LIN {X 0,Y 249.476,Z 748.518,A -85,B 0,C 180,E1 -18809.999,E2 -18809.999} C_VEL
LIN {X 0,Y 249.132,Z 748.626,A -85,B 0,C 180,E1 -18811.616,E2 -18811.616} C_VEL
LIN {X 0,Y 248.499,Z 747.93,A -85,B 0,C 180,E1 -18814.866,E2 -18814.866} C_VEL
LIN {X 0,Y 247.94,Z 746.023,A -85,B 0,C 180,E1 -18818.147,E2 -18818.147} C_VEL
LIN {X 0,Y 247.778,Z 742.93,A -85,B 0,C 180,E1 -18821.451,E2 -18821.451} C_VEL
LIN {X 0,Y 248.292,Z 738.587,A -85,B 0,C 180,E1 -18824.758,E2 -18824.758} C_VEL
LIN {X 0,Y 249.565,Z 732.939,A -85,B 0,C 180,E1 -18828.044,E2 -18828.044} C_VEL
LIN {X 0,Y 251.711,Z 725.892,A -85,B 0,C 180,E1 -18831.282,E2 -18831.282} C_VEL
LIN {X 0,Y 254.679,Z 717.261,A -85,B 0,C 180,E1 -18834.451,E2 -18834.451} C_VEL
LIN {X 0,Y 257.938,Z 708.169,A -85,B 0,C 180,E1 -18837.153,E2 -18837.153} C_VEL
LIN {X 0,Y 261.307,Z 699.031,A -85,B 0,C 180,E1 -18839.395,E2 -18839.395} C_VEL
LIN {X 0,Y 265.243,Z 688.365,A -85,B 0,C 180,E1 -18841.553,E2 -18841.553} C_VEL
LIN {X 0,Y 269.237,Z 676.854,A -85,B 0,C 180,E1 -18843.464,E2 -18843.464} C_VEL
LIN {X 0,Y 273.201,Z 664.412,A -85,B 0,C 180,E1 -18845.139,E2 -18845.139} C_VEL
LIN {X 0,Y 277.197,Z 650.888,A -85,B 0,C 180,E1 -18846.569,E2 -18846.569} C_VEL
LIN {X 0,Y 280.927,Z 635.963,A -85,B 0,C 180,E1 -18847.799,E2 -18847.799} C_VEL
LIN {X 0,Y 283.801,Z 621.53,A -85,B 0,C 180,E1 -18848.701,E2 -18848.701} C_VEL
LIN {X 0,Y 286.017,Z 605.972,A -85,B 0,C 180,E1 -18849.42,E2 -18849.42} C_VEL
LIN {X 0,Y 287.366,Z 589.732,A -85,B 0,C 180,E1 -18849.923,E2 -18849.923} C_VEL
LIN {X 0,Y 290.895,Z 520.508,A -85,B 0,C 180,E1 -18851.589,E2 -18851.589} C_VEL
LIN {X 0,Y 289.329,Z 502.503,A -85,B 0,C 180,E1 -18852.514,E2 -18852.514} C_VEL
LIN {X 0,Y 286.599,Z 477.609,A -85,B 0,C 180,E1 -18853.955,E2 -18853.955} C_VEL
LIN {X 0,Y 285.966,Z 473.872,A -85,B 0,C 180,E1 -18854.225,E2 -18854.225} C_VEL
LIN {X 0,Y 279.058,Z 458.877,A -85,B 0,C 180,E1 -18856.347,E2 -18856.347} C_VEL
LIN {X 0,Y 272.923,Z 447.108,A -85,B 0,C 180,E1 -18858.346,E2 -18858.346} C_VEL
LIN {X 0,Y 268.743,Z 439.718,A -85,B 0,C 180,E1 -18859.789,E2 -18859.789} C_VEL
LIN {X 0,Y 265.068,Z 433.428,A -85,B 0,C 180,E1 -18861.13,E2 -18861.13} C_VEL
LIN {X 0,Y 260.653,Z 426.199,A -85,B 0,C 180,E1 -18862.84,E2 -18862.84} C_VEL
LIN {X 0,Y 256.84,Z 420.001,A -85,B 0,C 180,E1 -18864.446,E2 -18864.446} C_VEL
LIN {X 0,Y 254.494,Z 413.539,A -85,B 0,C 180,E1 -18867.419,E2 -18867.419} C_VEL
LIN {X 0,Y 251.831,Z 406.905,A -85,B 0,C 180,E1 -18870.869,E2 -18870.869} C_VEL
LIN {X 0,Y 249.026,Z 400.088,A -85,B 0,C 180,E1 -18874.956,E2 -18874.956} C_VEL
LIN {X 0,Y 249.041,Z 400.084,A -85,B 0,C 180,E1 -18878.628,E2 -18878.628} C_VEL
LIN {X 0,Y 249.149,Z 400.073,A -85,B 0,C 180,E1 -18883.616,E2 -18883.616} C_VEL
LIN {X 0,Y 249.207,Z 400.066,A -85,B 0,C 180,E1 -18888.615,E2 -18888.615} C_VEL
LIN {X 0,Y 249.42,Z 400.043,A -85,B 0,C 180,E1 -18891.901,E2 -18891.901} C_VEL
LIN {X 0,Y 249.254,Z 400.062,A -85,B 0,C 180,E1 -18895.148,E2 -18895.148} C_VEL
LIN {X 0,Y 249.647,Z 400.005,A -85,B 0,C 180,E1 -18898.387,E2 -18898.387} C_VEL
LIN {X 0,Y 249.651,Z 400.002,A -85,B 0,C 180,E1 -18901.614,E2 -18901.614} C_VEL
LIN {X 0,Y 249.397,Z 399.996,A -85,B 0,C 180,E1 -18906.735,E2 -18906.735} C_VEL
LIN {X 0,Y 249.324,Z 400.04,A -85,B 0,C 180,E1 -18909.738,E2 -18909.738} C_VEL
LIN {X 0,Y 249.169,Z 400.033,A -85,B 0,C 180,E1 -18914.706,E2 -18914.706} C_VEL
LIN {X 0,Y 249.103,Z 400.079,A -85,B 0,C 180,E1 -18918.08,E2 -18918.08} C_VEL
LIN {X 0,Y 249.07,Z 400.051,A -85,B 0,C 180,E1 -18921.52,E2 -18921.52} C_VEL
LIN {X 0,Y 249.057,Z 400.222,A -85,B 0,C 180,E1 -18924.486,E2 -18924.486} C_VEL
LIN {X 0,Y 249.847,Z 402.583,A -85,B 0,C 180,E1 -18924.958,E2 -18924.958} C_VEL
LIN {X 0,Y 251.68,Z 404.775,A -85,B 0,C 180,E1 -18925.83,E2 -18925.83} C_VEL
LIN {X 0,Y 253.402,Z 405.892,A -85,B 0,C 180,E1 -18926.566,E2 -18926.566} C_VEL
LIN {X 0,Y 255.21,Z 409.013,A -85,B 0,C 180,E1 -18927.414,E2 -18927.414} C_VEL
LIN {X 0,Y 257.729,Z 411.478,A -85,B 0,C 180,E1 -18928.445,E2 -18928.445} C_VEL
LIN {X 0,Y 260.121,Z 414.887,A -85,B 0,C 180,E1 -18929.433,E2 -18929.433} C_VEL
LIN {X 0,Y 261.868,Z 416.787,A -85,B 0,C 180,E1 -18930.099,E2 -18930.099} C_VEL
LIN {X 0,Y 264.729,Z 420.479,A -85,B 0,C 180,E1 -18931.174,E2 -18931.174} C_VEL
LIN {X 0,Y 269.59,Z 427.111,A -85,B 0,C 180,E1 -18932.901,E2 -18932.901} C_VEL
LIN {X 0,Y 274.586,Z 434.03,A -85,B 0,C 180,E1 -18934.548,E2 -18934.548} C_VEL
LIN {X 0,Y 283.18,Z 447.173,A -85,B 0,C 180,E1 -18937.169,E2 -18937.169} C_VEL
LIN {X 0,Y 291.353,Z 460.987,A -85,B 0,C 180,E1 -18939.448,E2 -18939.448} C_VEL
LIN {X 0,Y 293.531,Z 464.988,A -85,B 0,C 180,E1 -18940.029,E2 -18940.029} C_VEL
LIN {X 0,Y 290.894,Z 517.972,A -85,B 0,C 180,E1 -18941.323,E2 -18941.323} C_VEL
LIN {X 0,Y 289.972,Z 539.395,A -85,B 0,C 180,E1 -18941.982,E2 -18941.982} C_VEL
LIN {X 0,Y 288.744,Z 554.324,A -85,B 0,C 180,E1 -18942.716,E2 -18942.716} C_VEL
LIN {X 0,Y 286.941,Z 567.715,A -85,B 0,C 180,E1 -18943.579,E2 -18943.579} C_VEL
LIN {X 0,Y 284.605,Z 581.657,A -85,B 0,C 180,E1 -18944.772,E2 -18944.772} C_VEL
LIN {X 0,Y 281.516,Z 595.873,A -85,B 0,C 180,E1 -18946.303,E2 -18946.303} C_VEL
LIN {X 0,Y 278.175,Z 608.428,A -85,B 0,C 180,E1 -18947.973,E2 -18947.973} C_VEL
LIN {X 0,Y 274.87,Z 619.546,A -85,B 0,C 180,E1 -18949.791,E2 -18949.791} C_VEL
LIN {X 0,Y 271.101,Z 630.65,A -85,B 0,C 180,E1 -18952,E2 -18952} C_VEL
LIN {X 0,Y 267.58,Z 639.923,A -85,B 0,C 180,E1 -18954.241,E2 -18954.241} C_VEL
LIN {X 0,Y 263.922,Z 648.935,A -85,B 0,C 180,E1 -18956.916,E2 -18956.916} C_VEL
LIN {X 0,Y 260.559,Z 656.451,A -85,B 0,C 180,E1 -18959.671,E2 -18959.671} C_VEL
LIN {X 0,Y 257.771,Z 662.395,A -85,B 0,C 180,E1 -18962.388,E2 -18962.388} C_VEL
LIN {X 0,Y 255.141,Z 667.863,A -85,B 0,C 180,E1 -18965.596,E2 -18965.596} C_VEL
LIN {X 0,Y 252.997,Z 671.949,A -85,B 0,C 180,E1 -18968.832,E2 -18968.832} C_VEL
LIN {X 0,Y 251.419,Z 674.771,A -85,B 0,C 180,E1 -18972.093,E2 -18972.093} C_VEL
LIN {X 0,Y 250.317,Z 676.423,A -85,B 0,C 180,E1 -18975.364,E2 -18975.364} C_VEL
LIN {X 0,Y 249.779,Z 676.905,A -85,B 0,C 180,E1 -18978.642,E2 -18978.642} C_VEL
LIN {X 0,Y 249.622,Z 676.258,A -85,B 0,C 180,E1 -18981.908,E2 -18981.908} C_VEL
LIN {X 0,Y 249.657,Z 674.55,A -85,B 0,C 180,E1 -18985.156,E2 -18985.156} C_VEL
LIN {X 0,Y 250.221,Z 671.7,A -85,B 0,C 180,E1 -18988.391,E2 -18988.391} C_VEL
LIN {X 0,Y 251.252,Z 667.656,A -85,B 0,C 180,E1 -18991.603,E2 -18991.603} C_VEL
LIN {X 0,Y 252.64,Z 662.347,A -85,B 0,C 180,E1 -18994.788,E2 -18994.788} C_VEL
LIN {X 0,Y 254.541,Z 655.601,A -85,B 0,C 180,E1 -18997.936,E2 -18997.936} C_VEL
LIN {X 0,Y 256.823,Z 647.225,A -85,B 0,C 180,E1 -19001.044,E2 -19001.044} C_VEL
LIN {X 0,Y 259.301,Z 638.318,A -85,B 0,C 180,E1 -19003.719,E2 -19003.719} C_VEL
LIN {X 0,Y 261.672,Z 629.26,A -85,B 0,C 180,E1 -19005.98,E2 -19005.98} C_VEL
LIN {X 0,Y 264.275,Z 618.53,A -85,B 0,C 180,E1 -19008.208,E2 -19008.208} C_VEL
LIN {X 0,Y 266.7,Z 606.853,A -85,B 0,C 180,E1 -19010.235,E2 -19010.235} C_VEL
LIN {X 0,Y 269.276,Z 594.003,A -85,B 0,C 180,E1 -19012.036,E2 -19012.036} C_VEL
LIN {X 0,Y 271.443,Z 581.475,A -85,B 0,C 180,E1 -19013.458,E2 -19013.458} C_VEL
LIN {X 0,Y 273.344,Z 567.926,A -85,B 0,C 180,E1 -19014.696,E2 -19014.696} C_VEL
LIN {X 0,Y 274.933,Z 552.816,A -85,B 0,C 180,E1 -19015.757,E2 -19015.757} C_VEL
LIN {X 0,Y 276.006,Z 537.572,A -85,B 0,C 180,E1 -19016.522,E2 -19016.522} C_VEL
LIN {X 0,Y 276.531,Z 519.72,A -85,B 0,C 180,E1 -19017.106,E2 -19017.106} C_VEL
LIN {X 0,Y 279.032,Z 452.977,A -85,B 0,C 180,E1 -19018.811,E2 -19018.811} C_VEL
LIN {X 0,Y 270.28,Z 435.589,A -85,B 0,C 180,E1 -19020.695,E2 -19020.695} C_VEL
LIN {X 0,Y 260.936,Z 419.389,A -85,B 0,C 180,E1 -19022.818,E2 -19022.818} C_VEL
LIN {X 0,Y 253.534,Z 407.906,A -85,B 0,C 180,E1 -19024.61,E2 -19024.61} C_VEL
LIN {X 0,Y 251.344,Z 404.489,A -85,B 0,C 180,E1 -19025.171,E2 -19025.171} C_VEL
LIN {X 0,Y 249.599,Z 402.156,A -85,B 0,C 180,E1 -19025.614,E2 -19025.614} C_VEL
LIN {X 0,Y 249.025,Z 400.089,A -85,B 0,C 180,E1 -19025.851,E2 -19025.851} C_VEL
LIN {X 0,Y 249.012,Z 400.093,A -85,B 0,C 180,E1 -19028.383,E2 -19028.383} C_VEL
LIN {X 0,Y 248.956,Z 400.094,A -85,B 0,C 180,E1 -19032.778,E2 -19032.778} C_VEL
LIN {X 0,Y 248.966,Z 400.089,A -85,B 0,C 180,E1 -19037.352,E2 -19037.352} C_VEL
LIN {X 0,Y 249.001,Z 400.085,A -85,B 0,C 180,E1 -19041.614,E2 -19041.614} C_VEL
LIN {X 0,Y 249.041,Z 400.079,A -85,B 0,C 180,E1 -19045.638,E2 -19045.638} C_VEL
LIN {X 0,Y 248.991,Z 400.093,A -85,B 0,C 180,E1 -19049.464,E2 -19049.464} C_VEL
LIN {X 0,Y 249.02,Z 400.093,A -85,B 0,C 180,E1 -19053.156,E2 -19053.156} C_VEL
LIN {X 0,Y 249.048,Z 400.077,A -85,B 0,C 180,E1 -19056.729,E2 -19056.729} C_VEL
LIN {X 0,Y 249.044,Z 400.08,A -85,B 0,C 180,E1 -19060.206,E2 -19060.206} C_VEL
LIN {X 0,Y 249.155,Z 400.076,A -85,B 0,C 180,E1 -19063.616,E2 -19063.616} C_VEL
LIN {X 0,Y 249.181,Z 400.035,A -85,B 0,C 180,E1 -19066.959,E2 -19066.959} C_VEL
LIN {X 0,Y 249.367,Z 399.996,A -85,B 0,C 180,E1 -19070.599,E2 -19070.599} C_VEL
LIN {X 0,Y 249.414,Z 400.036,A -85,B 0,C 180,E1 -19073.528,E2 -19073.528} C_VEL
LIN {X 0,Y 249.476,Z 400.016,A -85,B 0,C 180,E1 -19077.599,E2 -19077.599} C_VEL
LIN {X 0,Y 248.956,Z 400.086,A -85,B 0,C 180,E1 -19078.948,E2 -19078.948} C_VEL
LIN {X 0,Y 247.373,Z 400.295,A -85,B 0,C 180,E1 -19080.27,E2 -19080.27} C_VEL
LIN {X 0,Y 243.446,Z 400.774,A -85,B 0,C 180,E1 -19082.93,E2 -19082.93} C_VEL
LIN {X 0,Y 242.313,Z 400.91,A -85,B 0,C 180,E1 -19084.323,E2 -19084.323} C_VEL
LIN {X 0,Y 242.218,Z 400.925,A -85,B 0,C 180,E1 -19084.796,E2 -19084.796} C_VEL
LIN {X 0,Y 242.389,Z 400.915,A -85,B 0,C 180,E1 -19086.66,E2 -19086.66} C_VEL
LIN {X 0,Y 242.256,Z 400.921,A -85,B 0,C 180,E1 -19090.024,E2 -19090.024} C_VEL
LIN {X 0,Y 242.098,Z 400.944,A -85,B 0,C 180,E1 -19095.145,E2 -19095.145} C_VEL
LIN {X 0,Y 242.009,Z 400.954,A -85,B 0,C 180,E1 -19098.629,E2 -19098.629} C_VEL
LIN {X 0,Y 241.969,Z 400.963,A -85,B 0,C 180,E1 -19102.184,E2 -19102.184} C_VEL
LIN {X 0,Y 241.983,Z 400.962,A -85,B 0,C 180,E1 -19105.826,E2 -19105.826} C_VEL
LIN {X 0,Y 241.959,Z 400.966,A -85,B 0,C 180,E1 -19109.589,E2 -19109.589} C_VEL
LIN {X 0,Y 241.975,Z 400.948,A -85,B 0,C 180,E1 -19113.493,E2 -19113.493} C_VEL
LIN {X 0,Y 241.995,Z 401.064,A -85,B 0,C 180,E1 -19115.509,E2 -19115.509} C_VEL
LIN {X 0,Y 246.124,Z 413.213,A -85,B 0,C 180,E1 -19119.976,E2 -19119.976} C_VEL
LIN {X 0,Y 249.086,Z 422.878,A -85,B 0,C 180,E1 -19123.174,E2 -19123.174} C_VEL
LIN {X 0,Y 250.292,Z 426.911,A -85,B 0,C 180,E1 -19124.374,E2 -19124.374} C_VEL
LIN {X 0,Y 258.143,Z 443.198,A -85,B 0,C 180,E1 -19126.434,E2 -19126.434} C_VEL
LIN {X 0,Y 264.737,Z 458.633,A -85,B 0,C 180,E1 -19128.09,E2 -19128.09} C_VEL
LIN {X 0,Y 265.62,Z 461.45,A -85,B 0,C 180,E1 -19128.327,E2 -19128.327} C_VEL
LIN {X 0,Y 268.764,Z 492.72,A -85,B 0,C 180,E1 -19129.844,E2 -19129.844} C_VEL
LIN {X 0,Y 271.266,Z 519.191,A -85,B 0,C 180,E1 -19131.056,E2 -19131.056} C_VEL
LIN {X 0,Y 267.769,Z 598.776,A -85,B 0,C 180,E1 -19133.103,E2 -19133.103} C_VEL
LIN {X 0,Y 266.362,Z 614.419,A -85,B 0,C 180,E1 -19133.759,E2 -19133.759} C_VEL
LIN {X 0,Y 264.285,Z 629.484,A -85,B 0,C 180,E1 -19134.663,E2 -19134.663} C_VEL
LIN {X 0,Y 261.597,Z 644.604,A -85,B 0,C 180,E1 -19135.888,E2 -19135.888} C_VEL
LIN {X 0,Y 258.665,Z 657.774,A -85,B 0,C 180,E1 -19137.253,E2 -19137.253} C_VEL
LIN {X 0,Y 256.507,Z 666.573,A -85,B 0,C 180,E1 -19138.353,E2 -19138.353} C_VEL
LIN {X 0,Y 253.528,Z 679.329,A -85,B 0,C 180,E1 -19140.297,E2 -19140.297} C_VEL
LIN {X 0,Y 250.464,Z 690.836,A -85,B 0,C 180,E1 -19142.42,E2 -19142.42} C_VEL
LIN {X 0,Y 247.407,Z 702.532,A -85,B 0,C 180,E1 -19145.081,E2 -19145.081} C_VEL
LIN {X 0,Y 245.08,Z 711.881,A -85,B 0,C 180,E1 -19147.669,E2 -19147.669} C_VEL
LIN {X 0,Y 243.175,Z 720.586,A -85,B 0,C 180,E1 -19150.588,E2 -19150.588} C_VEL
LIN {X 0,Y 241.833,Z 727.828,A -85,B 0,C 180,E1 -19153.54,E2 -19153.54} C_VEL
LIN {X 0,Y 241.125,Z 733.822,A -85,B 0,C 180,E1 -19156.516,E2 -19156.516} C_VEL
LIN {X 0,Y 240.966,Z 739.281,A -85,B 0,C 180,E1 -19159.921,E2 -19159.921} C_VEL
LIN {X 0,Y 241.306,Z 743.356,A -85,B 0,C 180,E1 -19163.309,E2 -19163.309} C_VEL
LIN {X 0,Y 241.603,Z 744.896,A -85,B 0,C 180,E1 -19164.993,E2 -19164.993} C_VEL
LIN {X 0,Y 242.142,Z 746.94,A -85,B 0,C 180,E1 -19168.336,E2 -19168.336} C_VEL
LIN {X 0,Y 242.448,Z 747.474,A -85,B 0,C 180,E1 -19169.999,E2 -19169.999} C_VEL
LIN {X 0,Y 242.093,Z 747.598,A -85,B 0,C 180,E1 -19171.663,E2 -19171.663} C_VEL
LIN {X 0,Y 241.409,Z 746.93,A -85,B 0,C 180,E1 -19175.01,E2 -19175.01} C_VEL
LIN {X 0,Y 240.834,Z 745.054,A -85,B 0,C 180,E1 -19178.389,E2 -19178.389} C_VEL
LIN {X 0,Y 240.725,Z 741.993,A -85,B 0,C 180,E1 -19181.791,E2 -19181.791} C_VEL
LIN {X 0,Y 241.338,Z 737.677,A -85,B 0,C 180,E1 -19185.193,E2 -19185.193} C_VEL
LIN {X 0,Y 242.69,Z 732.068,A -85,B 0,C 180,E1 -19188.574,E2 -19188.574} C_VEL
LIN {X 0,Y 244.997,Z 725.073,A -85,B 0,C 180,E1 -19191.894,E2 -19191.894} C_VEL
LIN {X 0,Y 248.143,Z 716.501,A -85,B 0,C 180,E1 -19195.139,E2 -19195.139} C_VEL
LIN {X 0,Y 251.56,Z 707.476,A -85,B 0,C 180,E1 -19197.9,E2 -19197.9} C_VEL
LIN {X 0,Y 255.108,Z 698.413,A -85,B 0,C 180,E1 -19200.182,E2 -19200.182} C_VEL
LIN {X 0,Y 259.19,Z 687.83,A -85,B 0,C 180,E1 -19202.378,E2 -19202.378} C_VEL
LIN {X 0,Y 263.683,Z 675.235,A -85,B 0,C 180,E1 -19204.496,E2 -19204.496} C_VEL
LIN {X 0,Y 267.847,Z 662.7,A -85,B 0,C 180,E1 -19206.182,E2 -19206.182} C_VEL
LIN {X 0,Y 271.983,Z 649.046,A -85,B 0,C 180,E1 -19207.621,E2 -19207.621} C_VEL
LIN {X 0,Y 275.601,Z 634.964,A -85,B 0,C 180,E1 -19208.78,E2 -19208.78} C_VEL
LIN {X 0,Y 278.558,Z 620.543,A -85,B 0,C 180,E1 -19209.688,E2 -19209.688} C_VEL
LIN {X 0,Y 280.72,Z 605.925,A -85,B 0,C 180,E1 -19210.374,E2 -19210.374} C_VEL
LIN {X 0,Y 282.138,Z 590.291,A -85,B 0,C 180,E1 -19210.879,E2 -19210.879} C_VEL
LIN {X 0,Y 285.805,Z 521.741,A -85,B 0,C 180,E1 -19212.551,E2 -19212.551} C_VEL
LIN {X 0,Y 284.506,Z 505.394,A -85,B 0,C 180,E1 -19213.399,E2 -19213.399} C_VEL
LIN {X 0,Y 281.744,Z 479.095,A -85,B 0,C 180,E1 -19214.959,E2 -19214.959} C_VEL
LIN {X 0,Y 281.208,Z 476.865,A -85,B 0,C 180,E1 -19215.163,E2 -19215.163} C_VEL
LIN {X 0,Y 275.137,Z 463.465,A -85,B 0,C 180,E1 -19217.118,E2 -19217.118} C_VEL
LIN {X 0,Y 268.864,Z 451.319,A -85,B 0,C 180,E1 -19219.255,E2 -19219.255} C_VEL
LIN {X 0,Y 265.135,Z 444.539,A -85,B 0,C 180,E1 -19220.608,E2 -19220.608} C_VEL
LIN {X 0,Y 261.817,Z 438.739,A -85,B 0,C 180,E1 -19221.874,E2 -19221.874} C_VEL
LIN {X 0,Y 257.664,Z 431.782,A -85,B 0,C 180,E1 -19223.552,E2 -19223.552} C_VEL
LIN {X 0,Y 253.275,Z 424.794,A -85,B 0,C 180,E1 -19225.46,E2 -19225.46} C_VEL
LIN {X 0,Y 248.719,Z 417.542,A -85,B 0,C 180,E1 -19227.679,E2 -19227.679} C_VEL
LIN {X 0,Y 246.271,Z 411.332,A -85,B 0,C 180,E1 -19230.979,E2 -19230.979} C_VEL
LIN {X 0,Y 243.388,Z 404.393,A -85,B 0,C 180,E1 -19235.248,E2 -19235.248} C_VEL
LIN {X 0,Y 241.947,Z 401.013,A -85,B 0,C 180,E1 -19237.646,E2 -19237.646} C_VEL
LIN {X 0,Y 242.002,Z 400.965,A -85,B 0,C 180,E1 -19241.371,E2 -19241.371} C_VEL
LIN {X 0,Y 242.093,Z 400.954,A -85,B 0,C 180,E1 -19244.855,E2 -19244.855} C_VEL
LIN {X 0,Y 242.317,Z 400.917,A -85,B 0,C 180,E1 -19250.427,E2 -19250.427} C_VEL
LIN {X 0,Y 242.389,Z 400.906,A -85,B 0,C 180,E1 -19253.34,E2 -19253.34} C_VEL
LIN {X 0,Y 242.607,Z 400.882,A -85,B 0,C 180,E1 -19258.34,E2 -19258.34} C_VEL
LIN {X 0,Y 242.611,Z 400.878,A -85,B 0,C 180,E1 -19261.66,E2 -19261.66} C_VEL
LIN {X 0,Y 242.38,Z 400.87,A -85,B 0,C 180,E1 -19266.705,E2 -19266.705} C_VEL
LIN {X 0,Y 242.253,Z 400.925,A -85,B 0,C 180,E1 -19270.025,E2 -19270.025} C_VEL
LIN {X 0,Y 242.127,Z 400.911,A -85,B 0,C 180,E1 -19275.144,E2 -19275.144} C_VEL
LIN {X 0,Y 242.04,Z 400.947,A -85,B 0,C 180,E1 -19278.627,E2 -19278.627} C_VEL
LIN {X 0,Y 242.033,Z 400.966,A -85,B 0,C 180,E1 -19281.288,E2 -19281.288} C_VEL
LIN {X 0,Y 242.847,Z 403.534,A -85,B 0,C 180,E1 -19281.866,E2 -19281.866} C_VEL
LIN {X 0,Y 244.758,Z 405.758,A -85,B 0,C 180,E1 -19282.92,E2 -19282.92} C_VEL
LIN {X 0,Y 246.638,Z 406.982,A -85,B 0,C 180,E1 -19283.846,E2 -19283.846} C_VEL
LIN {X 0,Y 248.47,Z 410.136,A -85,B 0,C 180,E1 -19284.826,E2 -19284.826} C_VEL
LIN {X 0,Y 251.111,Z 412.591,A -85,B 0,C 180,E1 -19286.045,E2 -19286.045} C_VEL
LIN {X 0,Y 253.503,Z 415.98,A -85,B 0,C 180,E1 -19287.153,E2 -19287.153} C_VEL
LIN {X 0,Y 255.422,Z 418.046,A -85,B 0,C 180,E1 -19287.966,E2 -19287.966} C_VEL
LIN {X 0,Y 257.975,Z 421.43,A -85,B 0,C 180,E1 -19289.034,E2 -19289.034} C_VEL
LIN {X 0,Y 259.356,Z 423.134,A -85,B 0,C 180,E1 -19289.584,E2 -19289.584} C_VEL
LIN {X 0,Y 263.088,Z 428.119,A -85,B 0,C 180,E1 -19291.022,E2 -19291.022} C_VEL
LIN {X 0,Y 266.703,Z 433.046,A -85,B 0,C 180,E1 -19292.334,E2 -19292.334} C_VEL
LIN {X 0,Y 271.875,Z 440.463,A -85,B 0,C 180,E1 -19294.099,E2 -19294.099} C_VEL
LIN {X 0,Y 279.124,Z 451.673,A -85,B 0,C 180,E1 -19296.389,E2 -19296.389} C_VEL
LIN {X 0,Y 287.093,Z 465.293,A -85,B 0,C 180,E1 -19298.706,E2 -19298.706} C_VEL
LIN {X 0,Y 288.491,Z 467.862,A -85,B 0,C 180,E1 -19299.096,E2 -19299.096} C_VEL
LIN {X 0,Y 285.88,Z 517.389,A -85,B 0,C 180,E1 -19300.309,E2 -19300.309} C_VEL
LIN {X 0,Y 284.888,Z 539.899,A -85,B 0,C 180,E1 -19301.001,E2 -19301.001} C_VEL
LIN {X 0,Y 283.666,Z 554.622,A -85,B 0,C 180,E1 -19301.726,E2 -19301.726} C_VEL
LIN {X 0,Y 281.799,Z 568.179,A -85,B 0,C 180,E1 -19302.597,E2 -19302.597} C_VEL
LIN {X 0,Y 279.545,Z 581.338,A -85,B 0,C 180,E1 -19303.716,E2 -19303.716} C_VEL
LIN {X 0,Y 276.494,Z 595.225,A -85,B 0,C 180,E1 -19305.194,E2 -19305.194} C_VEL
LIN {X 0,Y 272.871,Z 608.583,A -85,B 0,C 180,E1 -19306.961,E2 -19306.961} C_VEL
LIN {X 0,Y 269.36,Z 619.805,A -85,B 0,C 180,E1 -19308.793,E2 -19308.793} C_VEL
LIN {X 0,Y 265.429,Z 631.04,A -85,B 0,C 180,E1 -19311.037,E2 -19311.037} C_VEL
LIN {X 0,Y 261.182,Z 641.842,A -85,B 0,C 180,E1 -19313.704,E2 -19313.704} C_VEL
LIN {X 0,Y 257.375,Z 650.701,A -85,B 0,C 180,E1 -19316.432,E2 -19316.432} C_VEL
LIN {X 0,Y 253.832,Z 658.261,A -85,B 0,C 180,E1 -19319.322,E2 -19319.322} C_VEL
LIN {X 0,Y 250.647,Z 664.691,A -85,B 0,C 180,E1 -19322.443,E2 -19322.443} C_VEL
LIN {X 0,Y 247.981,Z 669.856,A -85,B 0,C 180,E1 -19325.737,E2 -19325.737} C_VEL
LIN {X 0,Y 246.308,Z 672.817,A -85,B 0,C 180,E1 -19328.228,E2 -19328.228} C_VEL
LIN {X 0,Y 244.592,Z 675.7,A -85,B 0,C 180,E1 -19331.576,E2 -19331.576} C_VEL
LIN {X 0,Y 243.415,Z 677.401,A -85,B 0,C 180,E1 -19334.94,E2 -19334.94} C_VEL
LIN {X 0,Y 242.789,Z 677.917,A -85,B 0,C 180,E1 -19338.31,E2 -19338.31} C_VEL
LIN {X 0,Y 242.603,Z 677.323,A -85,B 0,C 180,E1 -19341.673,E2 -19341.673} C_VEL
LIN {X 0,Y 242.611,Z 675.672,A -85,B 0,C 180,E1 -19345.015,E2 -19345.015} C_VEL
LIN {X 0,Y 243.18,Z 672.879,A -85,B 0,C 180,E1 -19348.345,E2 -19348.345} C_VEL
LIN {X 0,Y 244.253,Z 668.892,A -85,B 0,C 180,E1 -19351.649,E2 -19351.649} C_VEL
LIN {X 0,Y 245.656,Z 663.651,A -85,B 0,C 180,E1 -19354.924,E2 -19354.924} C_VEL
LIN {X 0,Y 247.619,Z 656.972,A -85,B 0,C 180,E1 -19358.159,E2 -19358.159} C_VEL
LIN {X 0,Y 249.975,Z 648.679,A -85,B 0,C 180,E1 -19361.35,E2 -19361.35} C_VEL
LIN {X 0,Y 252.529,Z 639.858,A -85,B 0,C 180,E1 -19364.094,E2 -19364.094} C_VEL
LIN {X 0,Y 255.422,Z 629.232,A -85,B 0,C 180,E1 -19366.793,E2 -19366.793} C_VEL
LIN {X 0,Y 258.142,Z 618.335,A -85,B 0,C 180,E1 -19369.069,E2 -19369.069} C_VEL
LIN {X 0,Y 260.727,Z 606.417,A -85,B 0,C 180,E1 -19371.133,E2 -19371.133} C_VEL
LIN {X 0,Y 263.482,Z 593.234,A -85,B 0,C 180,E1 -19372.961,E2 -19372.961} C_VEL
LIN {X 0,Y 265.601,Z 580.35,A -85,B 0,C 180,E1 -19374.422,E2 -19374.422} C_VEL
LIN {X 0,Y 267.634,Z 566.182,A -85,B 0,C 180,E1 -19375.676,E2 -19375.676} C_VEL
LIN {X 0,Y 269.175,Z 551.454,A -85,B 0,C 180,E1 -19376.673,E2 -19376.673} C_VEL
LIN {X 0,Y 270.191,Z 536.263,A -85,B 0,C 180,E1 -19377.406,E2 -19377.406} C_VEL
LIN {X 0,Y 270.913,Z 511.116,A -85,B 0,C 180,E1 -19378.168,E2 -19378.168} C_VEL
LIN {X 0,Y 273.171,Z 455.24,A -85,B 0,C 180,E1 -19379.609,E2 -19379.609} C_VEL
LIN {X 0,Y 264.991,Z 438.961,A -85,B 0,C 180,E1 -19381.448,E2 -19381.448} C_VEL
LIN {X 0,Y 256.254,Z 423.785,A -85,B 0,C 180,E1 -19383.515,E2 -19383.515} C_VEL
LIN {X 0,Y 249.341,Z 412.874,A -85,B 0,C 180,E1 -19385.261,E2 -19385.261} C_VEL
LIN {X 0,Y 246.808,Z 409.184,A -85,B 0,C 180,E1 -19385.925,E2 -19385.925} C_VEL
LIN {X 0,Y 244.539,Z 405.59,A -85,B 0,C 180,E1 -19386.549,E2 -19386.549} C_VEL
LIN {X 0,Y 242.615,Z 403.171,A -85,B 0,C 180,E1 -19387.066,E2 -19387.066} C_VEL
LIN {X 0,Y 241.977,Z 400.963,A -85,B 0,C 180,E1 -19387.31,E2 -19387.31} C_VEL
LIN {X 0,Y 241.898,Z 400.979,A -85,B 0,C 180,E1 -19391.93,E2 -19391.93} C_VEL
LIN {X 0,Y 241.892,Z 400.974,A -85,B 0,C 180,E1 -19396.581,E2 -19396.581} C_VEL
LIN {X 0,Y 241.973,Z 400.96,A -85,B 0,C 180,E1 -19401.646,E2 -19401.646} C_VEL
LIN {X 0,Y 241.972,Z 400.971,A -85,B 0,C 180,E1 -19404.486,E2 -19404.486} C_VEL
LIN {X 0,Y 241.946,Z 400.974,A -85,B 0,C 180,E1 -19408.475,E2 -19408.475} C_VEL
LIN {X 0,Y 241.953,Z 400.969,A -85,B 0,C 180,E1 -19412.305,E2 -19412.305} C_VEL
LIN {X 0,Y 242.019,Z 400.95,A -85,B 0,C 180,E1 -19416.011,E2 -19416.011} C_VEL
LIN {X 0,Y 241.984,Z 400.963,A -85,B 0,C 180,E1 -19419.603,E2 -19419.603} C_VEL
LIN {X 0,Y 242.111,Z 400.951,A -85,B 0,C 180,E1 -19423.317,E2 -19423.317} C_VEL
LIN {X 0,Y 242.157,Z 400.888,A -85,B 0,C 180,E1 -19428.278,E2 -19428.278} C_VEL
LIN {X 0,Y 242.353,Z 400.886,A -85,B 0,C 180,E1 -19431.663,E2 -19431.663} C_VEL
LIN {X 0,Y 242.384,Z 400.91,A -85,B 0,C 180,E1 -19433.339,E2 -19433.339} C_VEL
LIN {X 0,Y 242.602,Z 400.872,A -85,B 0,C 180,E1 -19438.34,E2 -19438.34} C_VEL
LIN {X 0,Y 242.612,Z 400.885,A -85,B 0,C 180,E1 -19441.66,E2 -19441.66} C_VEL
LIN {X 0,Y 242.218,Z 400.925,A -85,B 0,C 180,E1 -19444.796,E2 -19444.796} C_VEL
LIN {X 0,Y 241.548,Z 401.021,A -85,B 0,C 180,E1 -19446.186,E2 -19446.186} C_VEL
LIN {X 0,Y 238.708,Z 401.391,A -85,B 0,C 180,E1 -19448.454,E2 -19448.454} C_VEL
LIN {X 0,Y 235.431,Z 401.792,A -85,B 0,C 180,E1 -19451.251,E2 -19451.251} C_VEL
LIN {X 0,Y 235.067,Z 401.827,A -85,B 0,C 180,E1 -19452.22,E2 -19452.22} C_VEL
LIN {X 0,Y 235.046,Z 401.833,A -85,B 0,C 180,E1 -19456.902,E2 -19456.902} C_VEL
LIN {X 0,Y 234.954,Z 401.838,A -85,B 0,C 180,E1 -19461.987,E2 -19461.987} C_VEL
LIN {X 0,Y 234.901,Z 401.843,A -85,B 0,C 180,E1 -19466.665,E2 -19466.665} C_VEL
LIN {X 0,Y 234.891,Z 401.851,A -85,B 0,C 180,E1 -19470.573,E2 -19470.573} C_VEL
LIN {X 0,Y 234.991,Z 402.02,A -85,B 0,C 180,E1 -19474.204,E2 -19474.204} C_VEL
LIN {X 0,Y 238.526,Z 412.295,A -85,B 0,C 180,E1 -19478.224,E2 -19478.224} C_VEL
LIN {X 0,Y 241.857,Z 422.842,A -85,B 0,C 180,E1 -19481.939,E2 -19481.939} C_VEL
LIN {X 0,Y 242.672,Z 425.504,A -85,B 0,C 180,E1 -19482.75,E2 -19482.75} C_VEL
LIN {X 0,Y 249.12,Z 438.303,A -85,B 0,C 180,E1 -19484.568,E2 -19484.568} C_VEL
LIN {X 0,Y 255.679,Z 452.618,A -85,B 0,C 180,E1 -19486.324,E2 -19486.324} C_VEL
LIN {X 0,Y 260.042,Z 463.529,A -85,B 0,C 180,E1 -19487.471,E2 -19487.471} C_VEL
LIN {X 0,Y 263.043,Z 494.261,A -85,B 0,C 180,E1 -19489.004,E2 -19489.004} C_VEL
LIN {X 0,Y 265.374,Z 520.907,A -85,B 0,C 180,E1 -19490.242,E2 -19490.242} C_VEL
LIN {X 0,Y 261.758,Z 598.911,A -85,B 0,C 180,E1 -19492.291,E2 -19492.291} C_VEL
LIN {X 0,Y 260.186,Z 614.929,A -85,B 0,C 180,E1 -19492.998,E2 -19492.998} C_VEL
LIN {X 0,Y 258.062,Z 629.621,A -85,B 0,C 180,E1 -19493.919,E2 -19493.919} C_VEL
LIN {X 0,Y 255.286,Z 644.456,A -85,B 0,C 180,E1 -19495.163,E2 -19495.163} C_VEL
LIN {X 0,Y 252.242,Z 657.712,A -85,B 0,C 180,E1 -19496.579,E2 -19496.579} C_VEL
LIN {X 0,Y 249.709,Z 667.784,A -85,B 0,C 180,E1 -19497.911,E2 -19497.911} C_VEL
LIN {X 0,Y 246.435,Z 681.046,A -85,B 0,C 180,E1 -19500.061,E2 -19500.061} C_VEL
LIN {X 0,Y 243.069,Z 693.032,A -85,B 0,C 180,E1 -19502.444,E2 -19502.444} C_VEL
LIN {X 0,Y 240.057,Z 704.136,A -85,B 0,C 180,E1 -19505.17,E2 -19505.17} C_VEL
LIN {X 0,Y 237.754,Z 713.14,A -85,B 0,C 180,E1 -19507.859,E2 -19507.859} C_VEL
LIN {X 0,Y 235.864,Z 721.479,A -85,B 0,C 180,E1 -19510.867,E2 -19510.867} C_VEL
LIN {X 0,Y 234.513,Z 729.3,A -85,B 0,C 180,E1 -19514.352,E2 -19514.352} C_VEL
LIN {X 0,Y 233.917,Z 735.534,A -85,B 0,C 180,E1 -19517.859,E2 -19517.859} C_VEL
LIN {X 0,Y 234.05,Z 740.349,A -85,B 0,C 180,E1 -19521.365,E2 -19521.365} C_VEL
LIN {X 0,Y 234.512,Z 743.794,A -85,B 0,C 180,E1 -19524.841,E2 -19524.841} C_VEL
LIN {X 0,Y 235.104,Z 745.873,A -85,B 0,C 180,E1 -19528.286,E2 -19528.286} C_VEL
LIN {X 0,Y 235.419,Z 746.428,A -85,B 0,C 180,E1 -19529.999,E2 -19529.999} C_VEL
LIN {X 0,Y 235.052,Z 746.57,A -85,B 0,C 180,E1 -19531.713,E2 -19531.713} C_VEL
LIN {X 0,Y 234.323,Z 745.931,A -85,B 0,C 180,E1 -19535.162,E2 -19535.162} C_VEL
LIN {X 0,Y 233.745,Z 744.087,A -85,B 0,C 180,E1 -19538.645,E2 -19538.645} C_VEL
LIN {X 0,Y 233.668,Z 741.046,A -85,B 0,C 180,E1 -19542.153,E2 -19542.153} C_VEL
LIN {X 0,Y 234.389,Z 736.766,A -85,B 0,C 180,E1 -19545.655,E2 -19545.655} C_VEL
LIN {X 0,Y 235.869,Z 731.205,A -85,B 0,C 180,E1 -19549.132,E2 -19549.132} C_VEL
LIN {X 0,Y 238.316,Z 724.261,A -85,B 0,C 180,E1 -19552.541,E2 -19552.541} C_VEL
LIN {X 0,Y 241.616,Z 715.742,A -85,B 0,C 180,E1 -19555.867,E2 -19555.867} C_VEL
LIN {X 0,Y 245.23,Z 706.782,A -85,B 0,C 180,E1 -19558.686,E2 -19558.686} C_VEL
LIN {X 0,Y 248.944,Z 697.793,A -85,B 0,C 180,E1 -19561.011,E2 -19561.011} C_VEL
LIN {X 0,Y 253.193,Z 687.295,A -85,B 0,C 180,E1 -19563.243,E2 -19563.243} C_VEL
LIN {X 0,Y 257.838,Z 674.805,A -85,B 0,C 180,E1 -19565.394,E2 -19565.394} C_VEL
LIN {X 0,Y 262.145,Z 662.38,A -85,B 0,C 180,E1 -19567.099,E2 -19567.099} C_VEL
LIN {X 0,Y 266.399,Z 648.875,A -85,B 0,C 180,E1 -19568.553,E2 -19568.553} C_VEL
LIN {X 0,Y 270.356,Z 633.986,A -85,B 0,C 180,E1 -19569.8,E2 -19569.8} C_VEL
LIN {X 0,Y 273.384,Z 619.589,A -85,B 0,C 180,E1 -19570.715,E2 -19570.715} C_VEL
LIN {X 0,Y 275.733,Z 604.109,A -85,B 0,C 180,E1 -19571.443,E2 -19571.443} C_VEL
LIN {X 0,Y 277.139,Z 588.34,A -85,B 0,C 180,E1 -19571.95,E2 -19571.95} C_VEL
LIN {X 0,Y 280.806,Z 522.801,A -85,B 0,C 180,E1 -19573.554,E2 -19573.554} C_VEL
LIN {X 0,Y 279.717,Z 507.921,A -85,B 0,C 180,E1 -19574.337,E2 -19574.337} C_VEL
LIN {X 0,Y 277.1,Z 481.838,A -85,B 0,C 180,E1 -19575.922,E2 -19575.922} C_VEL
LIN {X 0,Y 276.357,Z 479.536,A -85,B 0,C 180,E1 -19576.187,E2 -19576.187} C_VEL
LIN {X 0,Y 271.031,Z 467.673,A -85,B 0,C 180,E1 -19577.989,E2 -19577.989} C_VEL
LIN {X 0,Y 265.629,Z 456.871,A -85,B 0,C 180,E1 -19579.918,E2 -19579.918} C_VEL
LIN {X 0,Y 261.861,Z 449.873,A -85,B 0,C 180,E1 -19581.343,E2 -19581.343} C_VEL
LIN {X 0,Y 258.778,Z 444.354,A -85,B 0,C 180,E1 -19582.569,E2 -19582.569} C_VEL
LIN {X 0,Y 254.581,Z 437.141,A -85,B 0,C 180,E1 -19584.341,E2 -19584.341} C_VEL
LIN {X 0,Y 250.445,Z 430.423,A -85,B 0,C 180,E1 -19586.222,E2 -19586.222} C_VEL
LIN {X 0,Y 245.753,Z 423.018,A -85,B 0,C 180,E1 -19588.562,E2 -19588.562} C_VEL
LIN {X 0,Y 241.3,Z 416.59,A -85,B 0,C 180,E1 -19591.015,E2 -19591.015} C_VEL
LIN {X 0,Y 240.134,Z 414.556,A -85,B 0,C 180,E1 -19591.841,E2 -19591.841} C_VEL
LIN {X 0,Y 237.791,Z 408.686,A -85,B 0,C 180,E1 -19595.558,E2 -19595.558} C_VEL
LIN {X 0,Y 234.927,Z 401.852,A -85,B 0,C 180,E1 -19600.901,E2 -19600.901} C_VEL
LIN {X 0,Y 235.046,Z 401.836,A -85,B 0,C 180,E1 -19604.389,E2 -19604.389} C_VEL
LIN {X 0,Y 235.274,Z 401.794,A -85,B 0,C 180,E1 -19610.307,E2 -19610.307} C_VEL
LIN {X 0,Y 235.341,Z 401.785,A -85,B 0,C 180,E1 -19613.14,E2 -19613.14} C_VEL
LIN {X 0,Y 235.567,Z 401.758,A -85,B 0,C 180,E1 -19618.291,E2 -19618.291} C_VEL
LIN {X 0,Y 235.569,Z 401.755,A -85,B 0,C 180,E1 -19621.71,E2 -19621.71} C_VEL
LIN {X 0,Y 235.334,Z 401.746,A -85,B 0,C 180,E1 -19626.861,E2 -19626.861} C_VEL
LIN {X 0,Y 235.202,Z 401.809,A -85,B 0,C 180,E1 -19630.329,E2 -19630.329} C_VEL
LIN {X 0,Y 235.072,Z 401.793,A -85,B 0,C 180,E1 -19635.61,E2 -19635.61} C_VEL
LIN {X 0,Y 235.036,Z 401.831,A -85,B 0,C 180,E1 -19637.399,E2 -19637.399} C_VEL
LIN {X 0,Y 235.76,Z 404.268,A -85,B 0,C 180,E1 -19638.072,E2 -19638.072} C_VEL
LIN {X 0,Y 237.764,Z 406.637,A -85,B 0,C 180,E1 -19639.423,E2 -19639.423} C_VEL
LIN {X 0,Y 239.867,Z 407.873,A -85,B 0,C 180,E1 -19640.655,E2 -19640.655} C_VEL
LIN {X 0,Y 241.395,Z 410.809,A -85,B 0,C 180,E1 -19641.64,E2 -19641.64} C_VEL
LIN {X 0,Y 244.208,Z 413.221,A -85,B 0,C 180,E1 -19643.142,E2 -19643.142} C_VEL
LIN {X 0,Y 246.855,Z 417.077,A -85,B 0,C 180,E1 -19644.554,E2 -19644.554} C_VEL
LIN {X 0,Y 248.849,Z 419.059,A -85,B 0,C 180,E1 -19645.505,E2 -19645.505} C_VEL
LIN {X 0,Y 251.554,Z 422.634,A -85,B 0,C 180,E1 -19646.777,E2 -19646.777} C_VEL
LIN {X 0,Y 252.852,Z 424.155,A -85,B 0,C 180,E1 -19647.349,E2 -19647.349} C_VEL
LIN {X 0,Y 256.009,Z 428.128,A -85,B 0,C 180,E1 -19648.694,E2 -19648.694} C_VEL
LIN {X 0,Y 263.161,Z 437.985,A -85,B 0,C 180,E1 -19651.503,E2 -19651.503} C_VEL
LIN {X 0,Y 268.996,Z 446.53,A -85,B 0,C 180,E1 -19653.574,E2 -19653.574} C_VEL
LIN {X 0,Y 276.585,Z 458.582,A -85,B 0,C 180,E1 -19656.044,E2 -19656.044} C_VEL
LIN {X 0,Y 283.389,Z 470.562,A -85,B 0,C 180,E1 -19658.09,E2 -19658.09} C_VEL
LIN {X 0,Y 282.139,Z 493.284,A -85,B 0,C 180,E1 -19658.653,E2 -19658.653} C_VEL
LIN {X 0,Y 280.202,Z 535.236,A -85,B 0,C 180,E1 -19659.799,E2 -19659.799} C_VEL
LIN {X 0,Y 279.05,Z 550.553,A -85,B 0,C 180,E1 -19660.45,E2 -19660.45} C_VEL
LIN {X 0,Y 277.381,Z 564.741,A -85,B 0,C 180,E1 -19661.32,E2 -19661.32} C_VEL
LIN {X 0,Y 275.361,Z 576.859,A -85,B 0,C 180,E1 -19662.257,E2 -19662.257} C_VEL
LIN {X 0,Y 272.67,Z 589.986,A -85,B 0,C 180,E1 -19663.541,E2 -19663.541} C_VEL
LIN {X 0,Y 269.167,Z 603.5,A -85,B 0,C 180,E1 -19665.175,E2 -19665.175} C_VEL
LIN {X 0,Y 265.394,Z 615.775,A -85,B 0,C 180,E1 -19667.01,E2 -19667.01} C_VEL
LIN {X 0,Y 261.334,Z 627.553,A -85,B 0,C 180,E1 -19669.207,E2 -19669.207} C_VEL
LIN {X 0,Y 257.252,Z 637.945,A -85,B 0,C 180,E1 -19671.575,E2 -19671.575} C_VEL
LIN {X 0,Y 253.047,Z 647.669,A -85,B 0,C 180,E1 -19674.323,E2 -19674.323} C_VEL
LIN {X 0,Y 249.269,Z 655.687,A -85,B 0,C 180,E1 -19677.131,E2 -19677.131} C_VEL
LIN {X 0,Y 245.951,Z 662.24,A -85,B 0,C 180,E1 -19679.998,E2 -19679.998} C_VEL
LIN {X 0,Y 242.697,Z 668.363,A -85,B 0,C 180,E1 -19683.424,E2 -19683.424} C_VEL
LIN {X 0,Y 240.776,Z 671.747,A -85,B 0,C 180,E1 -19685.882,E2 -19685.882} C_VEL
LIN {X 0,Y 238.644,Z 675.309,A -85,B 0,C 180,E1 -19689.306,E2 -19689.306} C_VEL
LIN {X 0,Y 237.055,Z 677.653,A -85,B 0,C 180,E1 -19692.755,E2 -19692.755} C_VEL
LIN {X 0,Y 236.093,Z 678.786,A -85,B 0,C 180,E1 -19696.224,E2 -19696.224} C_VEL
LIN {X 0,Y 235.657,Z 678.779,A -85,B 0,C 180,E1 -19699.791,E2 -19699.791} C_VEL
LIN {X 0,Y 235.513,Z 677.729,A -85,B 0,C 180,E1 -19703.145,E2 -19703.145} C_VEL
LIN {X 0,Y 235.813,Z 675.566,A -85,B 0,C 180,E1 -19706.584,E2 -19706.584} C_VEL
LIN {X 0,Y 236.682,Z 672.236,A -85,B 0,C 180,E1 -19710.001,E2 -19710.001} C_VEL
LIN {X 0,Y 237.815,Z 667.712,A -85,B 0,C 180,E1 -19713.389,E2 -19713.389} C_VEL
LIN {X 0,Y 239.634,Z 661.808,A -85,B 0,C 180,E1 -19716.737,E2 -19716.737} C_VEL
LIN {X 0,Y 241.846,Z 654.437,A -85,B 0,C 180,E1 -19720.042,E2 -19720.042} C_VEL
LIN {X 0,Y 244.216,Z 646.54,A -85,B 0,C 180,E1 -19722.887,E2 -19722.887} C_VEL
LIN {X 0,Y 247.034,Z 637.074,A -85,B 0,C 180,E1 -19725.681,E2 -19725.681} C_VEL
LIN {X 0,Y 249.674,Z 627.424,A -85,B 0,C 180,E1 -19728.037,E2 -19728.037} C_VEL
LIN {X 0,Y 252.541,Z 615.977,A -85,B 0,C 180,E1 -19730.357,E2 -19730.357} C_VEL
LIN {X 0,Y 255.101,Z 604.604,A -85,B 0,C 180,E1 -19732.26,E2 -19732.26} C_VEL
LIN {X 0,Y 257.646,Z 592.335,A -85,B 0,C 180,E1 -19733.938,E2 -19733.938} C_VEL
LIN {X 0,Y 259.939,Z 579.029,A -85,B 0,C 180,E1 -19735.418,E2 -19735.418} C_VEL
LIN {X 0,Y 261.848,Z 565.468,A -85,B 0,C 180,E1 -19736.608,E2 -19736.608} C_VEL
LIN {X 0,Y 263.4,Z 550.622,A -85,B 0,C 180,E1 -19737.595,E2 -19737.595} C_VEL
LIN {X 0,Y 264.375,Z 535.49,A -85,B 0,C 180,E1 -19738.308,E2 -19738.308} C_VEL
LIN {X 0,Y 265.551,Z 499.93,A -85,B 0,C 180,E1 -19739.333,E2 -19739.333} C_VEL
LIN {X 0,Y 267.39,Z 457.609,A -85,B 0,C 180,E1 -19740.434,E2 -19740.434} C_VEL
LIN {X 0,Y 259.875,Z 442.629,A -85,B 0,C 180,E1 -19742.198,E2 -19742.198} C_VEL
LIN {X 0,Y 251.721,Z 428.259,A -85,B 0,C 180,E1 -19744.214,E2 -19744.214} C_VEL
LIN {X 0,Y 243.286,Z 414.922,A -85,B 0,C 180,E1 -19746.453,E2 -19746.453} C_VEL
LIN {X 0,Y 239.924,Z 410.217,A -85,B 0,C 180,E1 -19747.386,E2 -19747.386} C_VEL
LIN {X 0,Y 237.607,Z 406.561,A -85,B 0,C 180,E1 -19748.071,E2 -19748.071} C_VEL
LIN {X 0,Y 235.679,Z 404.259,A -85,B 0,C 180,E1 -19748.626,E2 -19748.626} C_VEL
LIN {X 0,Y 234.913,Z 401.845,A -85,B 0,C 180,E1 -19748.935,E2 -19748.935} C_VEL
LIN {X 0,Y 234.857,Z 401.847,A -85,B 0,C 180,E1 -19754.094,E2 -19754.094} C_VEL
LIN {X 0,Y 234.845,Z 401.855,A -85,B 0,C 180,E1 -19758.823,E2 -19758.823} C_VEL
LIN {X 0,Y 234.917,Z 401.841,A -85,B 0,C 180,E1 -19761.078,E2 -19761.078} C_VEL
LIN {X 0,Y 234.92,Z 401.84,A -85,B 0,C 180,E1 -19765.36,E2 -19765.36} C_VEL
LIN {X 0,Y 234.893,Z 401.849,A -85,B 0,C 180,E1 -19769.426,E2 -19769.426} C_VEL
LIN {X 0,Y 234.966,Z 401.843,A -85,B 0,C 180,E1 -19773.807,E2 -19773.807} C_VEL
LIN {X 0,Y 234.963,Z 401.843,A -85,B 0,C 180,E1 -19778.007,E2 -19778.007} C_VEL
LIN {X 0,Y 235.052,Z 401.828,A -85,B 0,C 180,E1 -19783.093,E2 -19783.093} C_VEL
LIN {X 0,Y 235.09,Z 401.771,A -85,B 0,C 180,E1 -19787.92,E2 -19787.92} C_VEL
LIN {X 0,Y 235.291,Z 401.759,A -85,B 0,C 180,E1 -19791.41,E2 -19791.41} C_VEL
LIN {X 0,Y 235.335,Z 401.786,A -85,B 0,C 180,E1 -19793.139,E2 -19793.139} C_VEL
LIN {X 0,Y 235.56,Z 401.749,A -85,B 0,C 180,E1 -19798.29,E2 -19798.29} C_VEL
LIN {X 0,Y 235.571,Z 401.762,A -85,B 0,C 180,E1 -19801.709,E2 -19801.709} C_VEL
LIN {X 0,Y 235.34,Z 401.794,A -85,B 0,C 180,E1 -19806.86,E2 -19806.86} C_VEL
LIN {X 0,Y 235.18,Z 401.804,A -85,B 0,C 180,E1 -19810.329,E2 -19810.329} C_VEL
LIN {X 0,Y 235.067,Z 401.827,A -85,B 0,C 180,E1 -19812.22,E2 -19812.22} C_VEL
LIN {X 0,Y 234.338,Z 401.91,A -85,B 0,C 180,E1 -19813.65,E2 -19813.65} C_VEL
LIN {X 0,Y 231.465,Z 402.276,A -85,B 0,C 180,E1 -19815.985,E2 -19815.985} C_VEL
LIN {X 0,Y 229.043,Z 402.58,A -85,B 0,C 180,E1 -19817.887,E2 -19817.887} C_VEL
LIN {X 0,Y 227.981,Z 402.708,A -85,B 0,C 180,E1 -19819.364,E2 -19819.364} C_VEL
LIN {X 0,Y 227.88,Z 402.717,A -85,B 0,C 180,E1 -19819.864,E2 -19819.864} C_VEL
LIN {X 0,Y 227.861,Z 402.72,A -85,B 0,C 180,E1 -19823.638,E2 -19823.638} C_VEL
LIN {X 0,Y 227.829,Z 402.729,A -85,B 0,C 180,E1 -19827.562,E2 -19827.562} C_VEL
LIN {X 0,Y 227.85,Z 402.726,A -85,B 0,C 180,E1 -19831.625,E2 -19831.625} C_VEL
LIN {X 0,Y 227.922,Z 402.827,A -85,B 0,C 180,E1 -19832.723,E2 -19832.723} C_VEL
LIN {X 0,Y 231.79,Z 413.966,A -85,B 0,C 180,E1 -19837.33,E2 -19837.33} C_VEL
LIN {X 0,Y 234.971,Z 423.914,A -85,B 0,C 180,E1 -19840.95,E2 -19840.95} C_VEL
LIN {X 0,Y 242.105,Z 437.614,A -85,B 0,C 180,E1 -19843.104,E2 -19843.104} C_VEL
LIN {X 0,Y 248.351,Z 450.871,A -85,B 0,C 180,E1 -19844.885,E2 -19844.885} C_VEL
LIN {X 0,Y 254.271,Z 465.107,A -85,B 0,C 180,E1 -19846.514,E2 -19846.514} C_VEL
LIN {X 0,Y 254.74,Z 467.699,A -85,B 0,C 180,E1 -19846.69,E2 -19846.69} C_VEL
LIN {X 0,Y 257.599,Z 498.295,A -85,B 0,C 180,E1 -19848.25,E2 -19848.25} C_VEL
LIN {X 0,Y 259.582,Z 520.508,A -85,B 0,C 180,E1 -19849.328,E2 -19849.328} C_VEL
LIN {X 0,Y 255.899,Z 597.781,A -85,B 0,C 180,E1 -19851.396,E2 -19851.396} C_VEL
LIN {X 0,Y 254.296,Z 613.847,A -85,B 0,C 180,E1 -19852.117,E2 -19852.117} C_VEL
LIN {X 0,Y 252.03,Z 628.527,A -85,B 0,C 180,E1 -19853.039,E2 -19853.039} C_VEL
LIN {X 0,Y 249.444,Z 642.481,A -85,B 0,C 180,E1 -19854.224,E2 -19854.224} C_VEL
LIN {X 0,Y 246.175,Z 656.365,A -85,B 0,C 180,E1 -19855.718,E2 -19855.718} C_VEL
LIN {X 0,Y 243.284,Z 667.39,A -85,B 0,C 180,E1 -19857.204,E2 -19857.204} C_VEL
LIN {X 0,Y 240.193,Z 679.443,A -85,B 0,C 180,E1 -19859.2,E2 -19859.2} C_VEL
LIN {X 0,Y 236.666,Z 691.521,A -85,B 0,C 180,E1 -19861.632,E2 -19861.632} C_VEL
LIN {X 0,Y 233.5,Z 702.653,A -85,B 0,C 180,E1 -19864.409,E2 -19864.409} C_VEL
LIN {X 0,Y 231.051,Z 711.773,A -85,B 0,C 180,E1 -19867.181,E2 -19867.181} C_VEL
LIN {X 0,Y 229.039,Z 720.176,A -85,B 0,C 180,E1 -19870.273,E2 -19870.273} C_VEL
LIN {X 0,Y 227.822,Z 726.324,A -85,B 0,C 180,E1 -19872.999,E2 -19872.999} C_VEL
LIN {X 0,Y 226.985,Z 732.905,A -85,B 0,C 180,E1 -19876.572,E2 -19876.572} C_VEL
LIN {X 0,Y 226.872,Z 738.093,A -85,B 0,C 180,E1 -19880.19,E2 -19880.19} C_VEL
LIN {X 0,Y 227.145,Z 741.115,A -85,B 0,C 180,E1 -19882.89,E2 -19882.89} C_VEL
LIN {X 0,Y 227.425,Z 742.685,A -85,B 0,C 180,E1 -19884.68,E2 -19884.68} C_VEL
LIN {X 0,Y 228.038,Z 744.802,A -85,B 0,C 180,E1 -19888.233,E2 -19888.233} C_VEL
LIN {X 0,Y 228.39,Z 745.382,A -85,B 0,C 180,E1 -19889.999,E2 -19889.999} C_VEL
LIN {X 0,Y 228.01,Z 745.541,A -85,B 0,C 180,E1 -19891.766,E2 -19891.766} C_VEL
LIN {X 0,Y 227.24,Z 744.931,A -85,B 0,C 180,E1 -19895.323,E2 -19895.323} C_VEL
LIN {X 0,Y 226.656,Z 743.119,A -85,B 0,C 180,E1 -19898.918,E2 -19898.918} C_VEL
LIN {X 0,Y 226.623,Z 740.094,A -85,B 0,C 180,E1 -19902.537,E2 -19902.537} C_VEL
LIN {X 0,Y 227.678,Z 734.863,A -85,B 0,C 180,E1 -19906.882,E2 -19906.882} C_VEL
LIN {X 0,Y 229.624,Z 728.793,A -85,B 0,C 180,E1 -19910.607,E2 -19910.607} C_VEL
LIN {X 0,Y 232.458,Z 721.531,A -85,B 0,C 180,E1 -19914.087,E2 -19914.087} C_VEL
LIN {X 0,Y 236.169,Z 712.637,A -85,B 0,C 180,E1 -19917.467,E2 -19917.467} C_VEL
LIN {X 0,Y 240.153,Z 703.297,A -85,B 0,C 180,E1 -19920.317,E2 -19920.317} C_VEL
LIN {X 0,Y 244.978,Z 692.18,A -85,B 0,C 180,E1 -19923.028,E2 -19923.028} C_VEL
LIN {X 0,Y 249.556,Z 680.892,A -85,B 0,C 180,E1 -19925.245,E2 -19925.245} C_VEL
LIN {X 0,Y 254.213,Z 668.466,A -85,B 0,C 180,E1 -19927.21,E2 -19927.21} C_VEL
LIN {X 0,Y 258.948,Z 654.961,A -85,B 0,C 180,E1 -19928.873,E2 -19928.873} C_VEL
LIN {X 0,Y 262.876,Z 641.763,A -85,B 0,C 180,E1 -19930.162,E2 -19930.162} C_VEL
LIN {X 0,Y 266.421,Z 627.417,A -85,B 0,C 180,E1 -19931.258,E2 -19931.258} C_VEL
LIN {X 0,Y 269.306,Z 612.713,A -85,B 0,C 180,E1 -19932.093,E2 -19932.093} C_VEL
LIN {X 0,Y 271.345,Z 597.763,A -85,B 0,C 180,E1 -19932.706,E2 -19932.706} C_VEL
LIN {X 0,Y 272.859,Z 576.912,A -85,B 0,C 180,E1 -19933.274,E2 -19933.274} C_VEL
LIN {X 0,Y 275.913,Z 523.161,A -85,B 0,C 180,E1 -19934.615,E2 -19934.615} C_VEL
LIN {X 0,Y 274.054,Z 499.669,A -85,B 0,C 180,E1 -19935.95,E2 -19935.95} C_VEL
LIN {X 0,Y 272.373,Z 484.018,A -85,B 0,C 180,E1 -19936.981,E2 -19936.981} C_VEL
LIN {X 0,Y 267.215,Z 472.224,A -85,B 0,C 180,E1 -19938.812,E2 -19938.812} C_VEL
LIN {X 0,Y 261.71,Z 461.033,A -85,B 0,C 180,E1 -19940.875,E2 -19940.875} C_VEL
LIN {X 0,Y 258.084,Z 454.176,A -85,B 0,C 180,E1 -19942.32,E2 -19942.32} C_VEL
LIN {X 0,Y 254.81,Z 448.312,A -85,B 0,C 180,E1 -19943.692,E2 -19943.692} C_VEL
LIN {X 0,Y 251.744,Z 442.852,A -85,B 0,C 180,E1 -19945.06,E2 -19945.06} C_VEL
LIN {X 0,Y 247.788,Z 436.254,A -85,B 0,C 180,E1 -19946.939,E2 -19946.939} C_VEL
LIN {X 0,Y 243.214,Z 428.845,A -85,B 0,C 180,E1 -19949.323,E2 -19949.323} C_VEL
LIN {X 0,Y 239.011,Z 422.558,A -85,B 0,C 180,E1 -19951.752,E2 -19951.752} C_VEL
LIN {X 0,Y 237.206,Z 419.925,A -85,B 0,C 180,E1 -19952.895,E2 -19952.895} C_VEL
LIN {X 0,Y 231.368,Z 411.207,A -85,B 0,C 180,E1 -19957.214,E2 -19957.214} C_VEL
LIN {X 0,Y 229.749,Z 407.337,A -85,B 0,C 180,E1 -19960.337,E2 -19960.337} C_VEL
LIN {X 0,Y 227.993,Z 402.71,A -85,B 0,C 180,E1 -19964.811,E2 -19964.811} C_VEL
LIN {X 0,Y 228.217,Z 402.673,A -85,B 0,C 180,E1 -19970.2,E2 -19970.2} C_VEL
LIN {X 0,Y 228.294,Z 402.664,A -85,B 0,C 180,E1 -19972.927,E2 -19972.927} C_VEL
LIN {X 0,Y 228.525,Z 402.635,A -85,B 0,C 180,E1 -19978.238,E2 -19978.238} C_VEL
LIN {X 0,Y 228.527,Z 402.633,A -85,B 0,C 180,E1 -19981.763,E2 -19981.763} C_VEL
LIN {X 0,Y 228.286,Z 402.623,A -85,B 0,C 180,E1 -19987.074,E2 -19987.074} C_VEL
LIN {X 0,Y 228.133,Z 402.693,A -85,B 0,C 180,E1 -19990.652,E2 -19990.652} C_VEL
LIN {X 0,Y 228.045,Z 402.801,A -85,B 0,C 180,E1 -19992.402,E2 -19992.402} C_VEL
LIN {X 0,Y 228.719,Z 405.003,A -85,B 0,C 180,E1 -19993.211,E2 -19993.211} C_VEL
LIN {X 0,Y 230.721,Z 407.416,A -85,B 0,C 180,E1 -19995.006,E2 -19995.006} C_VEL
LIN {X 0,Y 233.155,Z 408.878,A -85,B 0,C 180,E1 -19996.819,E2 -19996.819} C_VEL
LIN {X 0,Y 234.496,Z 411.556,A -85,B 0,C 180,E1 -19997.891,E2 -19997.891} C_VEL
LIN {X 0,Y 236.92,Z 413.876,A -85,B 0,C 180,E1 -19999.495,E2 -19999.495} C_VEL
LIN {X 0,Y 237.897,Z 414.572,A -85,B 0,C 180,E1 -20000.086,E2 -20000.086} C_VEL
LIN {X 0,Y 239.9,Z 417.809,A -85,B 0,C 180,E1 -20001.369,E2 -20001.369} C_VEL
LIN {X 0,Y 242.424,Z 420.164,A -85,B 0,C 180,E1 -20002.759,E2 -20002.759} C_VEL
LIN {X 0,Y 244.773,Z 423.495,A -85,B 0,C 180,E1 -20004.039,E2 -20004.039} C_VEL
LIN {X 0,Y 246.641,Z 425.514,A -85,B 0,C 180,E1 -20004.966,E2 -20004.966} C_VEL
LIN {X 0,Y 249.894,Z 429.552,A -85,B 0,C 180,E1 -20006.518,E2 -20006.518} C_VEL
LIN {X 0,Y 253.281,Z 434.064,A -85,B 0,C 180,E1 -20008.033,E2 -20008.033} C_VEL
LIN {X 0,Y 260.466,Z 444.102,A -85,B 0,C 180,E1 -20010.955,E2 -20010.955} C_VEL
LIN {X 0,Y 267.445,Z 454.637,A -85,B 0,C 180,E1 -20013.494,E2 -20013.494} C_VEL
LIN {X 0,Y 274.915,Z 467.122,A -85,B 0,C 180,E1 -20015.972,E2 -20015.972} C_VEL
LIN {X 0,Y 278.538,Z 473.655,A -85,B 0,C 180,E1 -20017.1,E2 -20017.1} C_VEL
LIN {X 0,Y 275.65,Z 527.519,A -85,B 0,C 180,E1 -20018.487,E2 -20018.487} C_VEL
LIN {X 0,Y 274.754,Z 544.217,A -85,B 0,C 180,E1 -20019.075,E2 -20019.075} C_VEL
LIN {X 0,Y 273.325,Z 558.585,A -85,B 0,C 180,E1 -20019.834,E2 -20019.834} C_VEL
LIN {X 0,Y 271.106,Z 572.767,A -85,B 0,C 180,E1 -20020.814,E2 -20020.814} C_VEL
LIN {X 0,Y 268.498,Z 586.173,A -85,B 0,C 180,E1 -20022.039,E2 -20022.039} C_VEL
LIN {X 0,Y 265.201,Z 599.523,A -85,B 0,C 180,E1 -20023.553,E2 -20023.553} C_VEL
LIN {X 0,Y 261.274,Z 612.446,A -85,B 0,C 180,E1 -20025.355,E2 -20025.355} C_VEL
LIN {X 0,Y 257.438,Z 623.794,A -85,B 0,C 180,E1 -20027.338,E2 -20027.338} C_VEL
LIN {X 0,Y 253.685,Z 633.554,A -85,B 0,C 180,E1 -20029.382,E2 -20029.382} C_VEL
LIN {X 0,Y 249.68,Z 642.844,A -85,B 0,C 180,E1 -20031.74,E2 -20031.74} C_VEL
LIN {X 0,Y 245.465,Z 651.882,A -85,B 0,C 180,E1 -20034.566,E2 -20034.566} C_VEL
LIN {X 0,Y 241.539,Z 659.533,A -85,B 0,C 180,E1 -20037.545,E2 -20037.545} C_VEL
LIN {X 0,Y 237.952,Z 666.164,A -85,B 0,C 180,E1 -20040.836,E2 -20040.836} C_VEL
LIN {X 0,Y 234.868,Z 671.555,A -85,B 0,C 180,E1 -20044.359,E2 -20044.359} C_VEL
LIN {X 0,Y 233.014,Z 674.554,A -85,B 0,C 180,E1 -20046.916,E2 -20046.916} C_VEL
LIN {X 0,Y 230.98,Z 677.639,A -85,B 0,C 180,E1 -20050.604,E2 -20050.604} C_VEL
LIN {X 0,Y 229.622,Z 679.32,A -85,B 0,C 180,E1 -20054.012,E2 -20054.012} C_VEL
LIN {X 0,Y 228.824,Z 679.942,A -85,B 0,C 180,E1 -20057.586,E2 -20057.586} C_VEL
LIN {X 0,Y 228.575,Z 679.453,A -85,B 0,C 180,E1 -20061.157,E2 -20061.157} C_VEL
LIN {X 0,Y 228.525,Z 677.915,A -85,B 0,C 180,E1 -20064.707,E2 -20064.707} C_VEL
LIN {X 0,Y 229.101,Z 675.234,A -85,B 0,C 180,E1 -20068.243,E2 -20068.243} C_VEL
LIN {X 0,Y 230.24,Z 671.343,A -85,B 0,C 180,E1 -20071.75,E2 -20071.75} C_VEL
LIN {X 0,Y 231.679,Z 666.203,A -85,B 0,C 180,E1 -20075.222,E2 -20075.222} C_VEL
LIN {X 0,Y 233.773,Z 659.654,A -85,B 0,C 180,E1 -20078.646,E2 -20078.646} C_VEL
LIN {X 0,Y 236.31,Z 651.536,A -85,B 0,C 180,E1 -20082.016,E2 -20082.016} C_VEL
LIN {X 0,Y 239.036,Z 642.859,A -85,B 0,C 180,E1 -20084.908,E2 -20084.908} C_VEL
LIN {X 0,Y 241.654,Z 634.041,A -85,B 0,C 180,E1 -20087.344,E2 -20087.344} C_VEL
LIN {X 0,Y 244.574,Z 623.652,A -85,B 0,C 180,E1 -20089.733,E2 -20089.733} C_VEL
LIN {X 0,Y 247.541,Z 611.263,A -85,B 0,C 180,E1 -20092.098,E2 -20092.098} C_VEL
LIN {X 0,Y 250.397,Z 598.715,A -85,B 0,C 180,E1 -20094.015,E2 -20094.015} C_VEL
LIN {X 0,Y 253.036,Z 584.906,A -85,B 0,C 180,E1 -20095.72,E2 -20095.72} C_VEL
LIN {X 0,Y 255.372,Z 570.351,A -85,B 0,C 180,E1 -20097.117,E2 -20097.117} C_VEL
LIN {X 0,Y 257.141,Z 555.199,A -85,B 0,C 180,E1 -20098.229,E2 -20098.229} C_VEL
LIN {X 0,Y 258.332,Z 539.82,A -85,B 0,C 180,E1 -20099.032,E2 -20099.032} C_VEL
LIN {X 0,Y 259.054,Z 518.682,A -85,B 0,C 180,E1 -20099.734,E2 -20099.734} C_VEL
LIN {X 0,Y 261.558,Z 459.788,A -85,B 0,C 180,E1 -20101.319,E2 -20101.319} C_VEL
LIN {X 0,Y 254.174,Z 445.032,A -85,B 0,C 180,E1 -20103.138,E2 -20103.138} C_VEL
LIN {X 0,Y 245.552,Z 429.975,A -85,B 0,C 180,E1 -20105.386,E2 -20105.386} C_VEL
LIN {X 0,Y 238.709,Z 419.309,A -85,B 0,C 180,E1 -20107.292,E2 -20107.292} C_VEL
LIN {X 0,Y 233.259,Z 411.412,A -85,B 0,C 180,E1 -20108.91,E2 -20108.91} C_VEL
LIN {X 0,Y 231.129,Z 408.084,A -85,B 0,C 180,E1 -20109.587,E2 -20109.587} C_VEL
LIN {X 0,Y 228.65,Z 405.346,A -85,B 0,C 180,E1 -20110.349,E2 -20110.349} C_VEL
LIN {X 0,Y 227.808,Z 402.726,A -85,B 0,C 180,E1 -20110.717,E2 -20110.717} C_VEL
LIN {X 0,Y 227.806,Z 402.733,A -85,B 0,C 180,E1 -20115.199,E2 -20115.199} C_VEL
LIN {X 0,Y 227.795,Z 402.738,A -85,B 0,C 180,E1 -20119.616,E2 -20119.616} C_VEL
LIN {X 0,Y 227.861,Z 402.729,A -85,B 0,C 180,E1 -20124.124,E2 -20124.124} C_VEL
LIN {X 0,Y 227.852,Z 402.73,A -85,B 0,C 180,E1 -20128.374,E2 -20128.374} C_VEL
LIN {X 0,Y 227.847,Z 402.726,A -85,B 0,C 180,E1 -20132.439,E2 -20132.439} C_VEL
LIN {X 0,Y 227.887,Z 402.711,A -85,B 0,C 180,E1 -20136.364,E2 -20136.364} C_VEL
LIN {X 0,Y 227.889,Z 402.714,A -85,B 0,C 180,E1 -20140.169,E2 -20140.169} C_VEL
LIN {X 0,Y 228.015,Z 402.708,A -85,B 0,C 180,E1 -20143.894,E2 -20143.894} C_VEL
LIN {X 0,Y 228.048,Z 402.651,A -85,B 0,C 180,E1 -20147.541,E2 -20147.541} C_VEL
LIN {X 0,Y 228.234,Z 402.631,A -85,B 0,C 180,E1 -20151.143,E2 -20151.143} C_VEL
LIN {X 0,Y 228.288,Z 402.66,A -85,B 0,C 180,E1 -20152.926,E2 -20152.926} C_VEL
LIN {X 0,Y 228.494,Z 402.628,A -85,B 0,C 180,E1 -20158.237,E2 -20158.237} C_VEL
LIN {X 0,Y 228.529,Z 402.639,A -85,B 0,C 180,E1 -20161.762,E2 -20161.762} C_VEL
LIN {X 0,Y 228.292,Z 402.672,A -85,B 0,C 180,E1 -20167.073,E2 -20167.073} C_VEL
LIN {X 0,Y 228.12,Z 402.686,A -85,B 0,C 180,E1 -20170.652,E2 -20170.652} C_VEL
LIN {X 0,Y 227.994,Z 402.709,A -85,B 0,C 180,E1 -20176.106,E2 -20176.106} C_VEL
LIN {X 0,Y 227.88,Z 402.717,A -85,B 0,C 180,E1 -20179.864,E2 -20179.864} C_VEL
LIN {X 0,Y 227.176,Z 402.813,A -85,B 0,C 180,E1 -20181.339,E2 -20181.339} C_VEL
LIN {X 0,Y 224.324,Z 403.161,A -85,B 0,C 180,E1 -20183.745,E2 -20183.745} C_VEL
LIN {X 0,Y 221.917,Z 403.462,A -85,B 0,C 180,E1 -20185.709,E2 -20185.709} C_VEL
LIN {X 0,Y 220.876,Z 403.592,A -85,B 0,C 180,E1 -20187.232,E2 -20187.232} C_VEL
LIN {X 0,Y 220.786,Z 403.602,A -85,B 0,C 180,E1 -20187.749,E2 -20187.749} C_VEL
LIN {X 0,Y 220.81,Z 403.65,A -85,B 0,C 180,E1 -20191.091,E2 -20191.091} C_VEL
LIN {X 0,Y 223.897,Z 412.182,A -85,B 0,C 180,E1 -20194.936,E2 -20194.936} C_VEL
LIN {X 0,Y 227.326,Z 422.406,A -85,B 0,C 180,E1 -20198.985,E2 -20198.985} C_VEL
LIN {X 0,Y 234.453,Z 435.724,A -85,B 0,C 180,E1 -20201.321,E2 -20201.321} C_VEL
LIN {X 0,Y 239.92,Z 446.799,A -85,B 0,C 180,E1 -20202.998,E2 -20202.998} C_VEL
LIN {X 0,Y 247.111,Z 463.13,A -85,B 0,C 180,E1 -20205.1,E2 -20205.1} C_VEL
LIN {X 0,Y 249.153,Z 468.434,A -85,B 0,C 180,E1 -20205.688,E2 -20205.688} C_VEL
LIN {X 0,Y 251.771,Z 497.018,A -85,B 0,C 180,E1 -20207.201,E2 -20207.201} C_VEL
LIN {X 0,Y 253.826,Z 522.011,A -85,B 0,C 180,E1 -20208.435,E2 -20208.435} C_VEL
LIN {X 0,Y 250.105,Z 596.617,A -85,B 0,C 180,E1 -20210.458,E2 -20210.458} C_VEL
LIN {X 0,Y 248.422,Z 612.727,A -85,B 0,C 180,E1 -20211.185,E2 -20211.185} C_VEL
LIN {X 0,Y 246.146,Z 627.459,A -85,B 0,C 180,E1 -20212.13,E2 -20212.13} C_VEL
LIN {X 0,Y 243.253,Z 642.344,A -85,B 0,C 180,E1 -20213.424,E2 -20213.424} C_VEL
LIN {X 0,Y 239.829,Z 656.279,A -85,B 0,C 180,E1 -20214.971,E2 -20214.971} C_VEL
LIN {X 0,Y 236.898,Z 666.996,A -85,B 0,C 180,E1 -20216.458,E2 -20216.458} C_VEL
LIN {X 0,Y 233.707,Z 678.945,A -85,B 0,C 180,E1 -20218.5,E2 -20218.5} C_VEL
LIN {X 0,Y 230.345,Z 690.017,A -85,B 0,C 180,E1 -20220.78,E2 -20220.78} C_VEL
LIN {X 0,Y 227.282,Z 700.309,A -85,B 0,C 180,E1 -20223.362,E2 -20223.362} C_VEL
LIN {X 0,Y 224.384,Z 710.406,A -85,B 0,C 180,E1 -20226.463,E2 -20226.463} C_VEL
LIN {X 0,Y 222.269,Z 718.876,A -85,B 0,C 180,E1 -20229.646,E2 -20229.646} C_VEL
LIN {X 0,Y 220.615,Z 726.799,A -85,B 0,C 180,E1 -20233.339,E2 -20233.339} C_VEL
LIN {X 0,Y 219.845,Z 733.137,A -85,B 0,C 180,E1 -20237.069,E2 -20237.069} C_VEL
LIN {X 0,Y 219.873,Z 738.052,A -85,B 0,C 180,E1 -20240.803,E2 -20240.803} C_VEL
LIN {X 0,Y 220.342,Z 741.567,A -85,B 0,C 180,E1 -20244.509,E2 -20244.509} C_VEL
LIN {X 0,Y 220.972,Z 743.73,A -85,B 0,C 180,E1 -20248.177,E2 -20248.177} C_VEL
LIN {X 0,Y 221.359,Z 744.337,A -85,B 0,C 180,E1 -20249.999,E2 -20249.999} C_VEL
LIN {X 0,Y 220.965,Z 744.512,A -85,B 0,C 180,E1 -20251.822,E2 -20251.822} C_VEL
LIN {X 0,Y 220.162,Z 743.933,A -85,B 0,C 180,E1 -20255.495,E2 -20255.495} C_VEL
LIN {X 0,Y 219.56,Z 742.15,A -85,B 0,C 180,E1 -20259.209,E2 -20259.209} C_VEL
LIN {X 0,Y 219.592,Z 739.144,A -85,B 0,C 180,E1 -20262.945,E2 -20262.945} C_VEL
LIN {X 0,Y 220.689,Z 734.293,A -85,B 0,C 180,E1 -20267.183,E2 -20267.183} C_VEL
LIN {X 0,Y 222.891,Z 727.947,A -85,B 0,C 180,E1 -20271.259,E2 -20271.259} C_VEL
LIN {X 0,Y 225.888,Z 720.727,A -85,B 0,C 180,E1 -20274.835,E2 -20274.835} C_VEL
LIN {X 0,Y 229.802,Z 711.906,A -85,B 0,C 180,E1 -20278.295,E2 -20278.295} C_VEL
LIN {X 0,Y 233.968,Z 702.614,A -85,B 0,C 180,E1 -20281.207,E2 -20281.207} C_VEL
LIN {X 0,Y 238.99,Z 691.583,A -85,B 0,C 180,E1 -20283.967,E2 -20283.967} C_VEL
LIN {X 0,Y 244.076,Z 679.625,A -85,B 0,C 180,E1 -20286.351,E2 -20286.351} C_VEL
LIN {X 0,Y 249.071,Z 666.867,A -85,B 0,C 180,E1 -20288.37,E2 -20288.37} C_VEL
LIN {X 0,Y 253.94,Z 653.238,A -85,B 0,C 180,E1 -20290.048,E2 -20290.048} C_VEL
LIN {X 0,Y 258.567,Z 638.014,A -85,B 0,C 180,E1 -20291.491,E2 -20291.491} C_VEL
LIN {X 0,Y 262.032,Z 624.168,A -85,B 0,C 180,E1 -20292.495,E2 -20292.495} C_VEL
LIN {X 0,Y 264.885,Z 608.679,A -85,B 0,C 180,E1 -20293.353,E2 -20293.353} C_VEL
LIN {X 0,Y 266.822,Z 593.92,A -85,B 0,C 180,E1 -20293.91,E2 -20293.91} C_VEL
LIN {X 0,Y 271.101,Z 523.747,A -85,B 0,C 180,E1 -20295.711,E2 -20295.711} C_VEL
LIN {X 0,Y 268.927,Z 495.892,A -85,B 0,C 180,E1 -20297.37,E2 -20297.37} C_VEL
LIN {X 0,Y 268.023,Z 487.453,A -85,B 0,C 180,E1 -20297.954,E2 -20297.954} C_VEL
LIN {X 0,Y 262.969,Z 475.794,A -85,B 0,C 180,E1 -20299.84,E2 -20299.84} C_VEL
LIN {X 0,Y 258.164,Z 465.799,A -85,B 0,C 180,E1 -20301.74,E2 -20301.74} C_VEL
LIN {X 0,Y 252.987,Z 455.752,A -85,B 0,C 180,E1 -20303.943,E2 -20303.943} C_VEL
LIN {X 0,Y 248.64,Z 448.03,A -85,B 0,C 180,E1 -20305.944,E2 -20305.944} C_VEL
LIN {X 0,Y 245.148,Z 442.028,A -85,B 0,C 180,E1 -20307.683,E2 -20307.683} C_VEL
LIN {X 0,Y 240.728,Z 434.696,A -85,B 0,C 180,E1 -20310.094,E2 -20310.094} C_VEL
LIN {X 0,Y 236.762,Z 428.497,A -85,B 0,C 180,E1 -20312.509,E2 -20312.509} C_VEL
LIN {X 0,Y 230.072,Z 418.429,A -85,B 0,C 180,E1 -20317.429,E2 -20317.429} C_VEL
LIN {X 0,Y 227.677,Z 415.172,A -85,B 0,C 180,E1 -20319.562,E2 -20319.562} C_VEL
LIN {X 0,Y 223.16,Z 407.901,A -85,B 0,C 180,E1 -20324.941,E2 -20324.941} C_VEL
LIN {X 0,Y 221.536,Z 405.602,A -85,B 0,C 180,E1 -20327.636,E2 -20327.636} C_VEL
LIN {X 0,Y 221.118,Z 403.637,A -85,B 0,C 180,E1 -20329.549,E2 -20329.549} C_VEL
LIN {X 0,Y 221.231,Z 403.545,A -85,B 0,C 180,E1 -20332.7,E2 -20332.7} C_VEL
LIN {X 0,Y 221.459,Z 403.514,A -85,B 0,C 180,E1 -20338.182,E2 -20338.182} C_VEL
LIN {X 0,Y 221.461,Z 403.513,A -85,B 0,C 180,E1 -20341.819,E2 -20341.819} C_VEL
LIN {X 0,Y 221.145,Z 403.674,A -85,B 0,C 180,E1 -20344.215,E2 -20344.215} C_VEL
LIN {X 0,Y 221.63,Z 405.459,A -85,B 0,C 180,E1 -20345.459,E2 -20345.459} C_VEL
LIN {X 0,Y 224.436,Z 408.674,A -85,B 0,C 180,E1 -20349.651,E2 -20349.651} C_VEL
LIN {X 0,Y 226.489,Z 409.718,A -85,B 0,C 180,E1 -20351.807,E2 -20351.807} C_VEL
LIN {X 0,Y 227.701,Z 412.4,A -85,B 0,C 180,E1 -20353.158,E2 -20353.158} C_VEL
LIN {X 0,Y 229.865,Z 414.602,A -85,B 0,C 180,E1 -20355.064,E2 -20355.064} C_VEL
LIN {X 0,Y 231.427,Z 415.584,A -85,B 0,C 180,E1 -20356.254,E2 -20356.254} C_VEL
LIN {X 0,Y 233.039,Z 418.443,A -85,B 0,C 180,E1 -20357.553,E2 -20357.553} C_VEL
LIN {X 0,Y 235.757,Z 420.885,A -85,B 0,C 180,E1 -20359.369,E2 -20359.369} C_VEL
LIN {X 0,Y 238.528,Z 424.866,A -85,B 0,C 180,E1 -20361.158,E2 -20361.158} C_VEL
LIN {X 0,Y 240.455,Z 426.808,A -85,B 0,C 180,E1 -20362.254,E2 -20362.254} C_VEL
LIN {X 0,Y 243.23,Z 430.445,A -85,B 0,C 180,E1 -20363.784,E2 -20363.784} C_VEL
LIN {X 0,Y 244.765,Z 432.35,A -85,B 0,C 180,E1 -20364.576,E2 -20364.576} C_VEL
LIN {X 0,Y 248.291,Z 437.013,A -85,B 0,C 180,E1 -20366.306,E2 -20366.306} C_VEL
LIN {X 0,Y 252.284,Z 442.415,A -85,B 0,C 180,E1 -20368.112,E2 -20368.112} C_VEL
LIN {X 0,Y 257.833,Z 450.314,A -85,B 0,C 180,E1 -20370.411,E2 -20370.411} C_VEL
LIN {X 0,Y 264.097,Z 459.972,A -85,B 0,C 180,E1 -20372.778,E2 -20372.778} C_VEL
LIN {X 0,Y 271.245,Z 472.124,A -85,B 0,C 180,E1 -20375.248,E2 -20375.248} C_VEL
LIN {X 0,Y 273.748,Z 476.677,A -85,B 0,C 180,E1 -20376.064,E2 -20376.064} C_VEL
LIN {X 0,Y 270.899,Z 527.08,A -85,B 0,C 180,E1 -20377.368,E2 -20377.368} C_VEL
LIN {X 0,Y 269.943,Z 544.604,A -85,B 0,C 180,E1 -20377.978,E2 -20377.978} C_VEL
LIN {X 0,Y 268.454,Z 559.182,A -85,B 0,C 180,E1 -20378.747,E2 -20378.747} C_VEL
LIN {X 0,Y 266.494,Z 571.693,A -85,B 0,C 180,E1 -20379.594,E2 -20379.594} C_VEL
LIN {X 0,Y 263.7,Z 585.912,A -85,B 0,C 180,E1 -20380.869,E2 -20380.869} C_VEL
LIN {X 0,Y 260.423,Z 598.983,A -85,B 0,C 180,E1 -20382.33,E2 -20382.33} C_VEL
LIN {X 0,Y 256.643,Z 611.433,A -85,B 0,C 180,E1 -20384.044,E2 -20384.044} C_VEL
LIN {X 0,Y 252.728,Z 622.674,A -85,B 0,C 180,E1 -20385.958,E2 -20385.958} C_VEL
LIN {X 0,Y 248.239,Z 633.943,A -85,B 0,C 180,E1 -20388.296,E2 -20388.296} C_VEL
LIN {X 0,Y 243.51,Z 644.543,A -85,B 0,C 180,E1 -20391.027,E2 -20391.027} C_VEL
LIN {X 0,Y 239.027,Z 653.666,A -85,B 0,C 180,E1 -20393.983,E2 -20393.983} C_VEL
LIN {X 0,Y 234.547,Z 661.891,A -85,B 0,C 180,E1 -20397.362,E2 -20397.362} C_VEL
LIN {X 0,Y 230.812,Z 668.402,A -85,B 0,C 180,E1 -20400.846,E2 -20400.846} C_VEL
LIN {X 0,Y 227.718,Z 673.425,A -85,B 0,C 180,E1 -20404.402,E2 -20404.402} C_VEL
LIN {X 0,Y 225.262,Z 677.101,A -85,B 0,C 180,E1 -20408.015,E2 -20408.015} C_VEL
LIN {X 0,Y 223.436,Z 679.512,A -85,B 0,C 180,E1 -20411.668,E2 -20411.668} C_VEL
LIN {X 0,Y 222.247,Z 680.753,A -85,B 0,C 180,E1 -20415.347,E2 -20415.347} C_VEL
LIN {X 0,Y 221.642,Z 680.823,A -85,B 0,C 180,E1 -20419.415,E2 -20419.415} C_VEL
LIN {X 0,Y 221.472,Z 679.912,A -85,B 0,C 180,E1 -20422.709,E2 -20422.709} C_VEL
LIN {X 0,Y 221.734,Z 677.862,A -85,B 0,C 180,E1 -20426.366,E2 -20426.366} C_VEL
LIN {X 0,Y 222.618,Z 674.623,A -85,B 0,C 180,E1 -20430.001,E2 -20430.001} C_VEL
LIN {X 0,Y 223.821,Z 670.184,A -85,B 0,C 180,E1 -20433.601,E2 -20433.601} C_VEL
LIN {X 0,Y 225.708,Z 664.412,A -85,B 0,C 180,E1 -20437.155,E2 -20437.155} C_VEL
LIN {X 0,Y 228.089,Z 657.179,A -85,B 0,C 180,E1 -20440.654,E2 -20440.654} C_VEL
LIN {X 0,Y 230.615,Z 649.442,A -85,B 0,C 180,E1 -20443.662,E2 -20443.662} C_VEL
LIN {X 0,Y 233.64,Z 640.152,A -85,B 0,C 180,E1 -20446.605,E2 -20446.605} C_VEL
LIN {X 0,Y 236.506,Z 630.703,A -85,B 0,C 180,E1 -20449.079,E2 -20449.079} C_VEL
LIN {X 0,Y 239.583,Z 619.508,A -85,B 0,C 180,E1 -20451.511,E2 -20451.511} C_VEL
LIN {X 0,Y 242.275,Z 608.467,A -85,B 0,C 180,E1 -20453.507,E2 -20453.507} C_VEL
LIN {X 0,Y 245.348,Z 595.06,A -85,B 0,C 180,E1 -20455.447,E2 -20455.447} C_VEL
LIN {X 0,Y 247.756,Z 581.963,A -85,B 0,C 180,E1 -20456.992,E2 -20456.992} C_VEL
LIN {X 0,Y 250.015,Z 567.403,A -85,B 0,C 180,E1 -20458.318,E2 -20458.318} C_VEL
LIN {X 0,Y 251.685,Z 552.676,A -85,B 0,C 180,E1 -20459.333,E2 -20459.333} C_VEL
LIN {X 0,Y 252.779,Z 537.389,A -85,B 0,C 180,E1 -20460.076,E2 -20460.076} C_VEL
LIN {X 0,Y 253.97,Z 503.848,A -85,B 0,C 180,E1 -20461.09,E2 -20461.09} C_VEL
LIN {X 0,Y 255.847,Z 462.032,A -85,B 0,C 180,E1 -20462.23,E2 -20462.23} C_VEL
LIN {X 0,Y 248.238,Z 446.961,A -85,B 0,C 180,E1 -20464.2,E2 -20464.2} C_VEL
LIN {X 0,Y 239.809,Z 432.302,A -85,B 0,C 180,E1 -20466.521,E2 -20466.521} C_VEL
LIN {X 0,Y 232.596,Z 421.197,A -85,B 0,C 180,E1 -20468.654,E2 -20468.654} C_VEL
LIN {X 0,Y 228.817,Z 415.851,A -85,B 0,C 180,E1 -20469.837,E2 -20469.837} C_VEL
LIN {X 0,Y 226.834,Z 412.985,A -85,B 0,C 180,E1 -20470.486,E2 -20470.486} C_VEL
LIN {X 0,Y 224.455,Z 409.751,A -85,B 0,C 180,E1 -20471.281,E2 -20471.281} C_VEL
LIN {X 0,Y 223.829,Z 408.62,A -85,B 0,C 180,E1 -20471.508,E2 -20471.508} C_VEL
LIN {X 0,Y 221.712,Z 406.421,A -85,B 0,C 180,E1 -20472.216,E2 -20472.216} C_VEL
LIN {X 0,Y 220.738,Z 403.608,A -85,B 0,C 180,E1 -20472.68,E2 -20472.68} C_VEL
LIN {X 0,Y 220.738,Z 403.605,A -85,B 0,C 180,E1 -20477.078,E2 -20477.078} C_VEL
LIN {X 0,Y 220.779,Z 403.606,A -85,B 0,C 180,E1 -20480.456,E2 -20480.456} C_VEL
LIN {X 0,Y 220.825,Z 403.598,A -85,B 0,C 180,E1 -20482.792,E2 -20482.792} C_VEL
LIN {X 0,Y 220.81,Z 403.598,A -85,B 0,C 180,E1 -20487.242,E2 -20487.242} C_VEL
LIN {X 0,Y 220.797,Z 403.596,A -85,B 0,C 180,E1 -20491.48,E2 -20491.48} C_VEL
LIN {X 0,Y 220.842,Z 403.588,A -85,B 0,C 180,E1 -20495.562,E2 -20495.562} C_VEL
LIN {X 0,Y 220.848,Z 403.596,A -85,B 0,C 180,E1 -20499.509,E2 -20499.509} C_VEL
LIN {X 0,Y 220.973,Z 403.584,A -85,B 0,C 180,E1 -20503.366,E2 -20503.366} C_VEL
LIN {X 0,Y 221.05,Z 403.51,A -85,B 0,C 180,E1 -20509.002,E2 -20509.002} C_VEL
LIN {X 0,Y 221.225,Z 403.533,A -85,B 0,C 180,E1 -20512.699,E2 -20512.699} C_VEL
LIN {X 0,Y 221.431,Z 403.508,A -85,B 0,C 180,E1 -20518.181,E2 -20518.181} C_VEL
LIN {X 0,Y 221.463,Z 403.518,A -85,B 0,C 180,E1 -20521.818,E2 -20521.818} C_VEL
LIN {X 0,Y 221.23,Z 403.549,A -85,B 0,C 180,E1 -20527.3,E2 -20527.3} C_VEL
LIN {X 0,Y 221.045,Z 403.571,A -85,B 0,C 180,E1 -20530.997,E2 -20530.997} C_VEL
LIN {X 0,Y 220.962,Z 403.588,A -85,B 0,C 180,E1 -20536.634,E2 -20536.634} C_VEL
LIN {X 0,Y 220.841,Z 403.601,A -85,B 0,C 180,E1 -20540.491,E2 -20540.491} C_VEL
LIN {X 0,Y 220.799,Z 403.607,A -85,B 0,C 180,E1 -20544.443,E2 -20544.443} C_VEL
LIN {X 0,Y 220.786,Z 403.602,A -85,B 0,C 180,E1 -20547.749,E2 -20547.749} C_VEL
LIN {X 0,Y 220.575,Z 403.981,A -85,B 0,C 180,E1 -20548.757,E2 -20548.757} C_VEL
LIN {X 0,Y 219.787,Z 405.661,A -85,B 0,C 180,E1 -20550.214,E2 -20550.214} C_VEL
LIN {X 0,Y 218.809,Z 408.239,A -85,B 0,C 180,E1 -20551.592,E2 -20551.592} C_VEL
LIN {X 0,Y 217.77,Z 413.629,A -85,B 0,C 180,E1 -20553.836,E2 -20553.836} C_VEL
LIN {X 0,Y 218.215,Z 416.892,A -85,B 0,C 180,E1 -20555.176,E2 -20555.176} C_VEL
LIN {X 0,Y 219.627,Z 420.934,A -85,B 0,C 180,E1 -20556.793,E2 -20556.793} C_VEL
LIN {X 0,Y 224.3,Z 429.312,A -85,B 0,C 180,E1 -20558.495,E2 -20558.495} C_VEL
LIN {X 0,Y 229.717,Z 439.31,A -85,B 0,C 180,E1 -20560.335,E2 -20560.335} C_VEL
LIN {X 0,Y 235.364,Z 450.953,A -85,B 0,C 180,E1 -20562.159,E2 -20562.159} C_VEL
LIN {X 0,Y 242.43,Z 467.425,A -85,B 0,C 180,E1 -20564.33,E2 -20564.33} C_VEL
LIN {X 0,Y 243.887,Z 471.578,A -85,B 0,C 180,E1 -20564.782,E2 -20564.782} C_VEL
LIN {X 0,Y 246.529,Z 502.44,A -85,B 0,C 180,E1 -20566.443,E2 -20566.443} C_VEL
LIN {X 0,Y 248.124,Z 522.91,A -85,B 0,C 180,E1 -20567.478,E2 -20567.478} C_VEL
LIN {X 0,Y 244.393,Z 595.418,A -85,B 0,C 180,E1 -20569.479,E2 -20569.479} C_VEL
LIN {X 0,Y 242.658,Z 611.598,A -85,B 0,C 180,E1 -20570.217,E2 -20570.217} C_VEL
LIN {X 0,Y 240.331,Z 626.368,A -85,B 0,C 180,E1 -20571.179,E2 -20571.179} C_VEL
LIN {X 0,Y 237.547,Z 640.334,A -85,B 0,C 180,E1 -20572.396,E2 -20572.396} C_VEL
LIN {X 0,Y 234.091,Z 653.974,A -85,B 0,C 180,E1 -20573.901,E2 -20573.901} C_VEL
LIN {X 0,Y 230.415,Z 667.152,A -85,B 0,C 180,E1 -20575.76,E2 -20575.76} C_VEL
LIN {X 0,Y 226.946,Z 679.54,A -85,B 0,C 180,E1 -20577.973,E2 -20577.973} C_VEL
LIN {X 0,Y 223.487,Z 690.346,A -85,B 0,C 180,E1 -20580.311,E2 -20580.311} C_VEL
LIN {X 0,Y 220.347,Z 700.416,A -85,B 0,C 180,E1 -20582.967,E2 -20582.967} C_VEL
LIN {X 0,Y 217.393,Z 710.331,A -85,B 0,C 180,E1 -20586.165,E2 -20586.165} C_VEL
LIN {X 0,Y 215.212,Z 718.631,A -85,B 0,C 180,E1 -20589.448,E2 -20589.448} C_VEL
LIN {X 0,Y 213.691,Z 725.545,A -85,B 0,C 180,E1 -20592.782,E2 -20592.782} C_VEL
LIN {X 0,Y 212.814,Z 731.935,A -85,B 0,C 180,E1 -20596.634,E2 -20596.634} C_VEL
LIN {X 0,Y 212.784,Z 736.892,A -85,B 0,C 180,E1 -20600.494,E2 -20600.494} C_VEL
LIN {X 0,Y 213.263,Z 740.447,A -85,B 0,C 180,E1 -20604.326,E2 -20604.326} C_VEL
LIN {X 0,Y 213.905,Z 742.658,A -85,B 0,C 180,E1 -20608.116,E2 -20608.116} C_VEL
LIN {X 0,Y 214.328,Z 743.291,A -85,B 0,C 180,E1 -20609.999,E2 -20609.999} C_VEL
LIN {X 0,Y 213.891,Z 743.479,A -85,B 0,C 180,E1 -20611.882,E2 -20611.882} C_VEL
LIN {X 0,Y 213.085,Z 742.936,A -85,B 0,C 180,E1 -20615.678,E2 -20615.678} C_VEL
LIN {X 0,Y 212.484,Z 741.175,A -85,B 0,C 180,E1 -20619.518,E2 -20619.518} C_VEL
LIN {X 0,Y 212.575,Z 738.194,A -85,B 0,C 180,E1 -20623.38,E2 -20623.38} C_VEL
LIN {X 0,Y 213.706,Z 733.695,A -85,B 0,C 180,E1 -20627.504,E2 -20627.504} C_VEL
LIN {X 0,Y 215.524,Z 728.622,A -85,B 0,C 180,E1 -20631.019,E2 -20631.019} C_VEL
LIN {X 0,Y 218.458,Z 721.829,A -85,B 0,C 180,E1 -20634.721,E2 -20634.721} C_VEL
LIN {X 0,Y 222.364,Z 713.485,A -85,B 0,C 180,E1 -20638.298,E2 -20638.298} C_VEL
LIN {X 0,Y 226.515,Z 704.718,A -85,B 0,C 180,E1 -20641.31,E2 -20641.31} C_VEL
LIN {X 0,Y 230.806,Z 695.939,A -85,B 0,C 180,E1 -20643.758,E2 -20643.758} C_VEL
LIN {X 0,Y 235.567,Z 685.616,A -85,B 0,C 180,E1 -20646.1,E2 -20646.1} C_VEL
LIN {X 0,Y 240.703,Z 673.433,A -85,B 0,C 180,E1 -20648.347,E2 -20648.347} C_VEL
LIN {X 0,Y 245.484,Z 661.338,A -85,B 0,C 180,E1 -20650.1,E2 -20650.1} C_VEL
LIN {X 0,Y 250.122,Z 648.303,A -85,B 0,C 180,E1 -20651.59,E2 -20651.59} C_VEL
LIN {X 0,Y 254.369,Z 634.076,A -85,B 0,C 180,E1 -20652.87,E2 -20652.87} C_VEL
LIN {X 0,Y 257.651,Z 620.664,A -85,B 0,C 180,E1 -20653.799,E2 -20653.799} C_VEL
LIN {X 0,Y 260.392,Z 605.986,A -85,B 0,C 180,E1 -20654.565,E2 -20654.565} C_VEL
LIN {X 0,Y 262.239,Z 590.41,A -85,B 0,C 180,E1 -20655.153,E2 -20655.153} C_VEL
LIN {X 0,Y 266.408,Z 524.839,A -85,B 0,C 180,E1 -20656.824,E2 -20656.824} C_VEL
LIN {X 0,Y 264.415,Z 497.731,A -85,B 0,C 180,E1 -20658.482,E2 -20658.482} C_VEL
LIN {X 0,Y 263.718,Z 490.768,A -85,B 0,C 180,E1 -20658.973,E2 -20658.973} C_VEL
LIN {X 0,Y 258.063,Z 477.569,A -85,B 0,C 180,E1 -20661.217,E2 -20661.217} C_VEL
LIN {X 0,Y 252.285,Z 465.754,A -85,B 0,C 180,E1 -20663.675,E2 -20663.675} C_VEL
LIN {X 0,Y 248.486,Z 458.486,A -85,B 0,C 180,E1 -20665.429,E2 -20665.429} C_VEL
LIN {X 0,Y 245.512,Z 453.054,A -85,B 0,C 180,E1 -20666.891,E2 -20666.891} C_VEL
LIN {X 0,Y 242.287,Z 447.35,A -85,B 0,C 180,E1 -20668.586,E2 -20668.586} C_VEL
LIN {X 0,Y 238.549,Z 440.938,A -85,B 0,C 180,E1 -20670.725,E2 -20670.725} C_VEL
LIN {X 0,Y 234.477,Z 434.314,A -85,B 0,C 180,E1 -20673.334,E2 -20673.334} C_VEL
LIN {X 0,Y 227.631,Z 423.655,A -85,B 0,C 180,E1 -20678.73,E2 -20678.73} C_VEL
LIN {X 0,Y 221.837,Z 414.601,A -85,B 0,C 180,E1 -20685.553,E2 -20685.553} C_VEL
LIN {X 0,Y 220.344,Z 412.161,A -85,B 0,C 180,E1 -20688.268,E2 -20688.268} C_VEL
LIN {X 0,Y 219.761,Z 410.572,A -85,B 0,C 180,E1 -20689.791,E2 -20689.791} C_VEL
LIN {X 0,Y 218.443,Z 409.948,A -85,B 0,C 180,E1 -20698.157,E2 -20698.157} C_VEL
LIN {X 0,Y 220.054,Z 410.645,A -85,B 0,C 180,E1 -20703.777,E2 -20703.777} C_VEL
LIN {X 0,Y 220.851,Z 412.918,A -85,B 0,C 180,E1 -20705.708,E2 -20705.708} C_VEL
LIN {X 0,Y 223.817,Z 415.948,A -85,B 0,C 180,E1 -20709.973,E2 -20709.973} C_VEL
LIN {X 0,Y 225.118,Z 416.732,A -85,B 0,C 180,E1 -20711.366,E2 -20711.366} C_VEL
LIN {X 0,Y 226.697,Z 419.69,A -85,B 0,C 180,E1 -20713.103,E2 -20713.103} C_VEL
LIN {X 0,Y 229.245,Z 421.907,A -85,B 0,C 180,E1 -20715.304,E2 -20715.304} C_VEL
LIN {X 0,Y 229.966,Z 422.751,A -85,B 0,C 180,E1 -20715.894,E2 -20715.894} C_VEL
LIN {X 0,Y 232.295,Z 426.125,A -85,B 0,C 180,E1 -20717.725,E2 -20717.725} C_VEL
LIN {X 0,Y 234.238,Z 427.909,A -85,B 0,C 180,E1 -20719.037,E2 -20719.037} C_VEL
LIN {X 0,Y 236.773,Z 431.49,A -85,B 0,C 180,E1 -20720.71,E2 -20720.71} C_VEL
LIN {X 0,Y 238.401,Z 433.212,A -85,B 0,C 180,E1 -20721.673,E2 -20721.673} C_VEL
LIN {X 0,Y 241.49,Z 437.171,A -85,B 0,C 180,E1 -20723.418,E2 -20723.418} C_VEL
LIN {X 0,Y 246.048,Z 443.359,A -85,B 0,C 180,E1 -20725.767,E2 -20725.767} C_VEL
LIN {X 0,Y 250.125,Z 449.014,A -85,B 0,C 180,E1 -20727.671,E2 -20727.671} C_VEL
LIN {X 0,Y 256.253,Z 457.918,A -85,B 0,C 180,E1 -20730.266,E2 -20730.266} C_VEL
LIN {X 0,Y 263.564,Z 469.909,A -85,B 0,C 180,E1 -20733.066,E2 -20733.066} C_VEL
LIN {X 0,Y 269.056,Z 479.74,A -85,B 0,C 180,E1 -20734.994,E2 -20734.994} C_VEL
LIN {X 0,Y 266.22,Z 527.411,A -85,B 0,C 180,E1 -20736.231,E2 -20736.231} C_VEL
LIN {X 0,Y 265.205,Z 545.451,A -85,B 0,C 180,E1 -20736.864,E2 -20736.864} C_VEL
LIN {X 0,Y 263.653,Z 560.104,A -85,B 0,C 180,E1 -20737.643,E2 -20737.643} C_VEL
LIN {X 0,Y 261.47,Z 573.475,A -85,B 0,C 180,E1 -20738.568,E2 -20738.568} C_VEL
LIN {X 0,Y 258.569,Z 587.44,A -85,B 0,C 180,E1 -20739.842,E2 -20739.842} C_VEL
LIN {X 0,Y 254.93,Z 601.224,A -85,B 0,C 180,E1 -20741.426,E2 -20741.426} C_VEL
LIN {X 0,Y 250.791,Z 613.975,A -85,B 0,C 180,E1 -20743.233,E2 -20743.233} C_VEL
LIN {X 0,Y 246.393,Z 625.928,A -85,B 0,C 180,E1 -20745.365,E2 -20745.365} C_VEL
LIN {X 0,Y 242.154,Z 636.057,A -85,B 0,C 180,E1 -20747.565,E2 -20747.565} C_VEL
LIN {X 0,Y 237.534,Z 645.884,A -85,B 0,C 180,E1 -20750.177,E2 -20750.177} C_VEL
LIN {X 0,Y 233.212,Z 654.262,A -85,B 0,C 180,E1 -20752.938,E2 -20752.938} C_VEL
LIN {X 0,Y 229.124,Z 661.539,A -85,B 0,C 180,E1 -20755.913,E2 -20755.913} C_VEL
LIN {X 0,Y 225.46,Z 667.646,A -85,B 0,C 180,E1 -20759.049,E2 -20759.049} C_VEL
LIN {X 0,Y 222.401,Z 672.504,A -85,B 0,C 180,E1 -20762.23,E2 -20762.23} C_VEL
LIN {X 0,Y 219.868,Z 676.282,A -85,B 0,C 180,E1 -20765.448,E2 -20765.448} C_VEL
LIN {X 0,Y 217.312,Z 679.691,A -85,B 0,C 180,E1 -20769.699,E2 -20769.699} C_VEL
LIN {X 0,Y 215.899,Z 681.234,A -85,B 0,C 180,E1 -20772.965,E2 -20772.965} C_VEL
LIN {X 0,Y 214.927,Z 681.965,A -85,B 0,C 180,E1 -20776.769,E2 -20776.769} C_VEL
LIN {X 0,Y 214.57,Z 681.583,A -85,B 0,C 180,E1 -20780.575,E2 -20780.575} C_VEL
LIN {X 0,Y 214.446,Z 680.155,A -85,B 0,C 180,E1 -20784.359,E2 -20784.359} C_VEL
LIN {X 0,Y 215.025,Z 677.556,A -85,B 0,C 180,E1 -20788.128,E2 -20788.128} C_VEL
LIN {X 0,Y 216.212,Z 673.747,A -85,B 0,C 180,E1 -20791.863,E2 -20791.863} C_VEL
LIN {X 0,Y 217.738,Z 668.73,A -85,B 0,C 180,E1 -20795.557,E2 -20795.557} C_VEL
LIN {X 0,Y 219.955,Z 662.315,A -85,B 0,C 180,E1 -20799.193,E2 -20799.193} C_VEL
LIN {X 0,Y 222.275,Z 655.434,A -85,B 0,C 180,E1 -20802.324,E2 -20802.324} C_VEL
LIN {X 0,Y 225.133,Z 647.153,A -85,B 0,C 180,E1 -20805.388,E2 -20805.388} C_VEL
LIN {X 0,Y 228.417,Z 637.203,A -85,B 0,C 180,E1 -20808.384,E2 -20808.384} C_VEL
LIN {X 0,Y 231.533,Z 627.047,A -85,B 0,C 180,E1 -20810.895,E2 -20810.895} C_VEL
LIN {X 0,Y 234.76,Z 614.93,A -85,B 0,C 180,E1 -20813.37,E2 -20813.37} C_VEL
LIN {X 0,Y 237.803,Z 602.747,A -85,B 0,C 180,E1 -20815.374,E2 -20815.374} C_VEL
LIN {X 0,Y 240.619,Z 589.432,A -85,B 0,C 180,E1 -20817.153,E2 -20817.153} C_VEL
LIN {X 0,Y 243.114,Z 575.592,A -85,B 0,C 180,E1 -20818.607,E2 -20818.607} C_VEL
LIN {X 0,Y 245.178,Z 560.649,A -85,B 0,C 180,E1 -20819.812,E2 -20819.812} C_VEL
LIN {X 0,Y 246.618,Z 545.883,A -85,B 0,C 180,E1 -20820.683,E2 -20820.683} C_VEL
LIN {X 0,Y 247.344,Z 530.439,A -85,B 0,C 180,E1 -20821.307,E2 -20821.307} C_VEL
LIN {X 0,Y 250.174,Z 464.293,A -85,B 0,C 180,E1 -20823.187,E2 -20823.187} C_VEL
LIN {X 0,Y 242.645,Z 449.473,A -85,B 0,C 180,E1 -20825.236,E2 -20825.236} C_VEL
LIN {X 0,Y 235.189,Z 436.468,A -85,B 0,C 180,E1 -20827.395,E2 -20827.395} C_VEL
LIN {X 0,Y 228.827,Z 426.498,A -85,B 0,C 180,E1 -20829.364,E2 -20829.364} C_VEL
LIN {X 0,Y 223.071,Z 418.271,A -85,B 0,C 180,E1 -20831.269,E2 -20831.269} C_VEL
LIN {X 0,Y 219.909,Z 413.905,A -85,B 0,C 180,E1 -20832.381,E2 -20832.381} C_VEL
LIN {X 0,Y 217.733,Z 411.024,A -85,B 0,C 180,E1 -20833.173,E2 -20833.173} C_VEL
LIN {X 0,Y 216.858,Z 409.544,A -85,B 0,C 180,E1 -20833.516,E2 -20833.516} C_VEL
LIN {X 0,Y 214.712,Z 407.355,A -85,B 0,C 180,E1 -20834.304,E2 -20834.304} C_VEL
LIN {X 0,Y 213.734,Z 404.688,A -85,B 0,C 180,E1 -20834.761,E2 -20834.761} C_VEL
LIN {X 0,Y 213.701,Z 404.487,A -85,B 0,C 180,E1 -20836.319,E2 -20836.319} C_VEL
LIN {X 0,Y 213.699,Z 404.491,A -85,B 0,C 180,E1 -20839.148,E2 -20839.148} C_VEL
LIN {X 0,Y 213.74,Z 404.489,A -85,B 0,C 180,E1 -20843.71,E2 -20843.71} C_VEL
LIN {X 0,Y 213.757,Z 404.486,A -85,B 0,C 180,E1 -20848.26,E2 -20848.26} C_VEL
LIN {X 0,Y 213.783,Z 404.479,A -85,B 0,C 180,E1 -20852.597,E2 -20852.597} C_VEL
LIN {X 0,Y 213.798,Z 404.469,A -85,B 0,C 180,E1 -20856.986,E2 -20856.986} C_VEL
LIN {X 0,Y 213.882,Z 404.464,A -85,B 0,C 180,E1 -20862.798,E2 -20862.798} C_VEL
LIN {X 0,Y 213.928,Z 404.421,A -85,B 0,C 180,E1 -20866.704,E2 -20866.704} C_VEL
LIN {X 0,Y 214.119,Z 404.378,A -85,B 0,C 180,E1 -20870.554,E2 -20870.554} C_VEL
LIN {X 0,Y 214.06,Z 404.446,A -85,B 0,C 180,E1 -20874.347,E2 -20874.347} C_VEL
LIN {X 0,Y 214.371,Z 404.386,A -85,B 0,C 180,E1 -20878.121,E2 -20878.121} C_VEL
LIN {X 0,Y 214.503,Z 404.385,A -85,B 0,C 180,E1 -20880,E2 -20880} C_VEL
LIN {X 0,Y 214.399,Z 404.398,A -85,B 0,C 180,E1 -20881.878,E2 -20881.878} C_VEL
LIN {X 0,Y 214.171,Z 404.426,A -85,B 0,C 180,E1 -20887.542,E2 -20887.542} C_VEL
LIN {X 0,Y 213.978,Z 404.454,A -85,B 0,C 180,E1 -20891.365,E2 -20891.365} C_VEL
LIN {X 0,Y 213.86,Z 404.46,A -85,B 0,C 180,E1 -20895.242,E2 -20895.242} C_VEL
LIN {X 0,Y 213.785,Z 404.47,A -85,B 0,C 180,E1 -20899.192,E2 -20899.192} C_VEL
LIN {X 0,Y 213.781,Z 404.472,A -85,B 0,C 180,E1 -20903.234,E2 -20903.234} C_VEL
LIN {X 0,Y 213.756,Z 404.483,A -85,B 0,C 180,E1 -20908.471,E2 -20908.471} C_VEL
LIN {X 0,Y 213.775,Z 404.657,A -85,B 0,C 180,E1 -20909.411,E2 -20909.411} C_VEL
LIN {X 0,Y 217.264,Z 414.008,A -85,B 0,C 180,E1 -20913.917,E2 -20913.917} C_VEL
LIN {X 0,Y 218.215,Z 416.892,A -85,B 0,C 180,E1 -20915.176,E2 -20915.176} C_VEL
LIN {X 0,Y 218.898,Z 419.291,A -85,B 0,C 180,E1 -20915.96,E2 -20915.96} C_VEL
LIN {X 0,Y 219.925,Z 423.917,A -85,B 0,C 180,E1 -20916.875,E2 -20916.875} C_VEL
LIN {X 0,Y 220.962,Z 429.151,A -85,B 0,C 180,E1 -20917.568,E2 -20917.568} C_VEL
LIN {X 0,Y 222.667,Z 436.493,A -85,B 0,C 180,E1 -20918.383,E2 -20918.383} C_VEL
LIN {X 0,Y 224.419,Z 441.625,A -85,B 0,C 180,E1 -20919.086,E2 -20919.086} C_VEL
LIN {X 0,Y 225.182,Z 443.171,A -85,B 0,C 180,E1 -20919.356,E2 -20919.356} C_VEL
LIN {X 0,Y 232.369,Z 458.487,A -85,B 0,C 180,E1 -20921.784,E2 -20921.784} C_VEL
LIN {X 0,Y 238.636,Z 473.907,A -85,B 0,C 180,E1 -20923.795,E2 -20923.795} C_VEL
LIN {X 0,Y 242.516,Z 522.341,A -85,B 0,C 180,E1 -20926.426,E2 -20926.426} C_VEL
LIN {X 0,Y 238.763,Z 594.215,A -85,B 0,C 180,E1 -20928.455,E2 -20928.455} C_VEL
LIN {X 0,Y 236.954,Z 610.463,A -85,B 0,C 180,E1 -20929.199,E2 -20929.199} C_VEL
LIN {X 0,Y 234.563,Z 625.266,A -85,B 0,C 180,E1 -20930.176,E2 -20930.176} C_VEL
LIN {X 0,Y 231.471,Z 640.185,A -85,B 0,C 180,E1 -20931.507,E2 -20931.507} C_VEL
LIN {X 0,Y 227.914,Z 653.683,A -85,B 0,C 180,E1 -20933.037,E2 -20933.037} C_VEL
LIN {X 0,Y 224.27,Z 666.129,A -85,B 0,C 180,E1 -20934.834,E2 -20934.834} C_VEL
LIN {X 0,Y 220.845,Z 677.922,A -85,B 0,C 180,E1 -20936.977,E2 -20936.977} C_VEL
LIN {X 0,Y 217.246,Z 688.828,A -85,B 0,C 180,E1 -20939.368,E2 -20939.368} C_VEL
LIN {X 0,Y 213.927,Z 698.975,A -85,B 0,C 180,E1 -20942.086,E2 -20942.086} C_VEL
LIN {X 0,Y 210.786,Z 708.958,A -85,B 0,C 180,E1 -20945.369,E2 -20945.369} C_VEL
LIN {X 0,Y 208.444,Z 717.32,A -85,B 0,C 180,E1 -20948.749,E2 -20948.749} C_VEL
LIN {X 0,Y 206.783,Z 724.289,A -85,B 0,C 180,E1 -20952.188,E2 -20952.188} C_VEL
LIN {X 0,Y 205.798,Z 730.73,A -85,B 0,C 180,E1 -20956.169,E2 -20956.169} C_VEL
LIN {X 0,Y 205.684,Z 735.719,A -85,B 0,C 180,E1 -20960.163,E2 -20960.163} C_VEL
LIN {X 0,Y 206.19,Z 739.327,A -85,B 0,C 180,E1 -20964.13,E2 -20964.13} C_VEL
LIN {X 0,Y 206.837,Z 741.585,A -85,B 0,C 180,E1 -20968.052,E2 -20968.052} C_VEL
LIN {X 0,Y 207.293,Z 742.243,A -85,B 0,C 180,E1 -20969.999,E2 -20969.999} C_VEL
LIN {X 0,Y 206.817,Z 742.445,A -85,B 0,C 180,E1 -20971.947,E2 -20971.947} C_VEL
LIN {X 0,Y 206.007,Z 741.938,A -85,B 0,C 180,E1 -20975.873,E2 -20975.873} C_VEL
LIN {X 0,Y 205.411,Z 740.191,A -85,B 0,C 180,E1 -20979.849,E2 -20979.849} C_VEL
LIN {X 0,Y 205.569,Z 737.246,A -85,B 0,C 180,E1 -20983.845,E2 -20983.845} C_VEL
LIN {X 0,Y 206.746,Z 733.084,A -85,B 0,C 180,E1 -20987.86,E2 -20987.86} C_VEL
LIN {X 0,Y 208.805,Z 727.767,A -85,B 0,C 180,E1 -20991.729,E2 -20991.729} C_VEL
LIN {X 0,Y 211.921,Z 721.024,A -85,B 0,C 180,E1 -20995.537,E2 -20995.537} C_VEL
LIN {X 0,Y 215.472,Z 713.898,A -85,B 0,C 180,E1 -20998.755,E2 -20998.755} C_VEL
LIN {X 0,Y 219.744,Z 705.387,A -85,B 0,C 180,E1 -21001.849,E2 -21001.849} C_VEL
LIN {X 0,Y 224.904,Z 695.299,A -85,B 0,C 180,E1 -21004.769,E2 -21004.769} C_VEL
LIN {X 0,Y 229.83,Z 685.058,A -85,B 0,C 180,E1 -21007.15,E2 -21007.15} C_VEL
LIN {X 0,Y 235.146,Z 672.977,A -85,B 0,C 180,E1 -21009.426,E2 -21009.426} C_VEL
LIN {X 0,Y 240.098,Z 661.008,A -85,B 0,C 180,E1 -21011.191,E2 -21011.191} C_VEL
LIN {X 0,Y 244.867,Z 648.132,A -85,B 0,C 180,E1 -21012.691,E2 -21012.691} C_VEL
LIN {X 0,Y 249.224,Z 634.126,A -85,B 0,C 180,E1 -21013.978,E2 -21013.978} C_VEL
LIN {X 0,Y 252.589,Z 621.05,A -85,B 0,C 180,E1 -21014.91,E2 -21014.91} C_VEL
LIN {X 0,Y 255.544,Z 606.097,A -85,B 0,C 180,E1 -21015.711,E2 -21015.711} C_VEL
LIN {X 0,Y 257.519,Z 590.58,A -85,B 0,C 180,E1 -21016.317,E2 -21016.317} C_VEL
LIN {X 0,Y 261.813,Z 525.969,A -85,B 0,C 180,E1 -21017.977,E2 -21017.977} C_VEL
LIN {X 0,Y 259.917,Z 498.34,A -85,B 0,C 180,E1 -21019.713,E2 -21019.713} C_VEL
LIN {X 0,Y 259.484,Z 494.146,A -85,B 0,C 180,E1 -21020.028,E2 -21020.028} C_VEL
LIN {X 0,Y 254.372,Z 481.98,A -85,B 0,C 180,E1 -21022.171,E2 -21022.171} C_VEL
LIN {X 0,Y 248.831,Z 470.31,A -85,B 0,C 180,E1 -21024.665,E2 -21024.665} C_VEL
LIN {X 0,Y 243.666,Z 460.129,A -85,B 0,C 180,E1 -21027.234,E2 -21027.234} C_VEL
LIN {X 0,Y 239.655,Z 452.992,A -85,B 0,C 180,E1 -21029.414,E2 -21029.414} C_VEL
LIN {X 0,Y 236.204,Z 446.843,A -85,B 0,C 180,E1 -21031.495,E2 -21031.495} C_VEL
LIN {X 0,Y 232.317,Z 440.28,A -85,B 0,C 180,E1 -21034.118,E2 -21034.118} C_VEL
LIN {X 0,Y 226.098,Z 430.256,A -85,B 0,C 180,E1 -21039.264,E2 -21039.264} C_VEL
LIN {X 0,Y 220.683,Z 421.458,A -85,B 0,C 180,E1 -21045.947,E2 -21045.947} C_VEL
LIN {X 0,Y 219.235,Z 418.938,A -85,B 0,C 180,E1 -21048.75,E2 -21048.75} C_VEL
LIN {X 0,Y 218.739,Z 417.558,A -85,B 0,C 180,E1 -21050.143,E2 -21050.143} C_VEL
LIN {X 0,Y 217.882,Z 417.079,A -85,B 0,C 180,E1 -21060,E2 -21060} C_VEL
LIN {X 0,Y 219.016,Z 417.715,A -85,B 0,C 180,E1 -21063.45,E2 -21063.45} C_VEL
LIN {X 0,Y 219.969,Z 420.079,A -85,B 0,C 180,E1 -21065.731,E2 -21065.731} C_VEL
LIN {X 0,Y 222.704,Z 422.896,A -85,B 0,C 180,E1 -21069.727,E2 -21069.727} C_VEL
LIN {X 0,Y 223.781,Z 423.625,A -85,B 0,C 180,E1 -21070.926,E2 -21070.926} C_VEL
LIN {X 0,Y 225.479,Z 426.656,A -85,B 0,C 180,E1 -21072.832,E2 -21072.832} C_VEL
LIN {X 0,Y 228.281,Z 429.253,A -85,B 0,C 180,E1 -21075.299,E2 -21075.299} C_VEL
LIN {X 0,Y 230.702,Z 432.8,A -85,B 0,C 180,E1 -21077.273,E2 -21077.273} C_VEL
LIN {X 0,Y 232.471,Z 434.563,A -85,B 0,C 180,E1 -21078.519,E2 -21078.519} C_VEL
LIN {X 0,Y 235.237,Z 438.295,A -85,B 0,C 180,E1 -21080.381,E2 -21080.381} C_VEL
LIN {X 0,Y 236.68,Z 440.108,A -85,B 0,C 180,E1 -21081.274,E2 -21081.274} C_VEL
LIN {X 0,Y 240.577,Z 445.233,A -85,B 0,C 180,E1 -21083.513,E2 -21083.513} C_VEL
LIN {X 0,Y 246.084,Z 452.816,A -85,B 0,C 180,E1 -21086.325,E2 -21086.325} C_VEL
LIN {X 0,Y 253.247,Z 463.486,A -85,B 0,C 180,E1 -21089.537,E2 -21089.537} C_VEL
LIN {X 0,Y 259.856,Z 474.567,A -85,B 0,C 180,E1 -21092.187,E2 -21092.187} C_VEL
LIN {X 0,Y 264.438,Z 482.914,A -85,B 0,C 180,E1 -21093.883,E2 -21093.883} C_VEL
LIN {X 0,Y 261.971,Z 522.283,A -85,B 0,C 180,E1 -21094.905,E2 -21094.905} C_VEL
LIN {X 0,Y 260.729,Z 544.568,A -85,B 0,C 180,E1 -21095.635,E2 -21095.635} C_VEL
LIN {X 0,Y 259.232,Z 559.069,A -85,B 0,C 180,E1 -21096.376,E2 -21096.376} C_VEL
LIN {X 0,Y 257.37,Z 570.576,A -85,B 0,C 180,E1 -21097.126,E2 -21097.126} C_VEL
LIN {X 0,Y 254.405,Z 585.211,A -85,B 0,C 180,E1 -21098.387,E2 -21098.387} C_VEL
LIN {X 0,Y 250.794,Z 599.221,A -85,B 0,C 180,E1 -21099.938,E2 -21099.938} C_VEL
LIN {X 0,Y 246.782,Z 611.721,A -85,B 0,C 180,E1 -21101.643,E2 -21101.643} C_VEL
LIN {X 0,Y 242.532,Z 623.194,A -85,B 0,C 180,E1 -21103.58,E2 -21103.58} C_VEL
LIN {X 0,Y 237.652,Z 634.721,A -85,B 0,C 180,E1 -21105.979,E2 -21105.979} C_VEL
LIN {X 0,Y 233.067,Z 644.326,A -85,B 0,C 180,E1 -21108.443,E2 -21108.443} C_VEL
LIN {X 0,Y 228.153,Z 653.646,A -85,B 0,C 180,E1 -21111.41,E2 -21111.41} C_VEL
LIN {X 0,Y 223.6,Z 661.513,A -85,B 0,C 180,E1 -21114.558,E2 -21114.558} C_VEL
LIN {X 0,Y 219.318,Z 668.388,A -85,B 0,C 180,E1 -21118.081,E2 -21118.081} C_VEL
LIN {X 0,Y 215.859,Z 673.561,A -85,B 0,C 180,E1 -21121.532,E2 -21121.532} C_VEL
LIN {X 0,Y 213.326,Z 677.126,A -85,B 0,C 180,E1 -21124.643,E2 -21124.643} C_VEL
LIN {X 0,Y 210.508,Z 680.714,A -85,B 0,C 180,E1 -21129.199,E2 -21129.199} C_VEL
LIN {X 0,Y 209.059,Z 682.192,A -85,B 0,C 180,E1 -21132.39,E2 -21132.39} C_VEL
LIN {X 0,Y 207.976,Z 682.979,A -85,B 0,C 180,E1 -21136.318,E2 -21136.318} C_VEL
LIN {X 0,Y 207.574,Z 682.648,A -85,B 0,C 180,E1 -21140.255,E2 -21140.255} C_VEL
LIN {X 0,Y 207.409,Z 681.27,A -85,B 0,C 180,E1 -21144.166,E2 -21144.166} C_VEL
LIN {X 0,Y 207.988,Z 678.7,A -85,B 0,C 180,E1 -21148.064,E2 -21148.064} C_VEL
LIN {X 0,Y 209.195,Z 674.949,A -85,B 0,C 180,E1 -21151.926,E2 -21151.926} C_VEL
LIN {X 0,Y 210.76,Z 669.994,A -85,B 0,C 180,E1 -21155.742,E2 -21155.742} C_VEL
LIN {X 0,Y 213.039,Z 663.648,A -85,B 0,C 180,E1 -21159.495,E2 -21159.495} C_VEL
LIN {X 0,Y 215.857,Z 655.75,A -85,B 0,C 180,E1 -21163.174,E2 -21163.174} C_VEL
LIN {X 0,Y 218.866,Z 647.325,A -85,B 0,C 180,E1 -21166.318,E2 -21166.318} C_VEL
LIN {X 0,Y 222.331,Z 637.206,A -85,B 0,C 180,E1 -21169.385,E2 -21169.385} C_VEL
LIN {X 0,Y 225.589,Z 626.855,A -85,B 0,C 180,E1 -21171.953,E2 -21171.953} C_VEL
LIN {X 0,Y 228.697,Z 615.628,A -85,B 0,C 180,E1 -21174.269,E2 -21174.269} C_VEL
LIN {X 0,Y 231.868,Z 603.375,A -85,B 0,C 180,E1 -21176.314,E2 -21176.314} C_VEL
LIN {X 0,Y 234.803,Z 589.966,A -85,B 0,C 180,E1 -21178.126,E2 -21178.126} C_VEL
LIN {X 0,Y 237.393,Z 575.994,A -85,B 0,C 180,E1 -21179.606,E2 -21179.606} C_VEL
LIN {X 0,Y 239.448,Z 561.583,A -85,B 0,C 180,E1 -21180.784,E2 -21180.784} C_VEL
LIN {X 0,Y 240.969,Z 546.764,A -85,B 0,C 180,E1 -21181.667,E2 -21181.667} C_VEL
LIN {X 0,Y 241.707,Z 531.765,A -85,B 0,C 180,E1 -21182.29,E2 -21182.29} C_VEL
LIN {X 0,Y 244.211,Z 477.297,A -85,B 0,C 180,E1 -21183.853,E2 -21183.853} C_VEL
LIN {X 0,Y 244.585,Z 466.557,A -85,B 0,C 180,E1 -21184.186,E2 -21184.186} C_VEL
LIN {X 0,Y 236.769,Z 451.29,A -85,B 0,C 180,E1 -21186.429,E2 -21186.429} C_VEL
LIN {X 0,Y 229.307,Z 438.362,A -85,B 0,C 180,E1 -21188.724,E2 -21188.724} C_VEL
LIN {X 0,Y 221.525,Z 426.546,A -85,B 0,C 180,E1 -21191.314,E2 -21191.314} C_VEL
LIN {X 0,Y 216.197,Z 419.163,A -85,B 0,C 180,E1 -21193.238,E2 -21193.238} C_VEL
LIN {X 0,Y 213.298,Z 415.147,A -85,B 0,C 180,E1 -21194.358,E2 -21194.358} C_VEL
LIN {X 0,Y 210.958,Z 412.151,A -85,B 0,C 180,E1 -21195.292,E2 -21195.292} C_VEL
LIN {X 0,Y 210.063,Z 410.572,A -85,B 0,C 180,E1 -21195.683,E2 -21195.683} C_VEL
LIN {X 0,Y 207.843,Z 408.526,A -85,B 0,C 180,E1 -21196.578,E2 -21196.578} C_VEL
LIN {X 0,Y 206.786,Z 406.278,A -85,B 0,C 180,E1 -21197.089,E2 -21197.089} C_VEL
LIN {X 0,Y 206.616,Z 405.363,A -85,B 0,C 180,E1 -21197.225,E2 -21197.225} C_VEL
LIN {X 0,Y 206.667,Z 405.357,A -85,B 0,C 180,E1 -21201.457,E2 -21201.457} C_VEL
LIN {X 0,Y 206.699,Z 405.361,A -85,B 0,C 180,E1 -21204.688,E2 -21204.688} C_VEL
LIN {X 0,Y 206.694,Z 405.362,A -85,B 0,C 180,E1 -21209.334,E2 -21209.334} C_VEL
LIN {X 0,Y 206.701,Z 405.364,A -85,B 0,C 180,E1 -21213.767,E2 -21213.767} C_VEL
LIN {X 0,Y 206.715,Z 405.361,A -85,B 0,C 180,E1 -21218.038,E2 -21218.038} C_VEL
LIN {X 0,Y 206.801,Z 405.339,A -85,B 0,C 180,E1 -21222.19,E2 -21222.19} C_VEL
LIN {X 0,Y 206.869,Z 405.309,A -85,B 0,C 180,E1 -21226.242,E2 -21226.242} C_VEL
LIN {X 0,Y 207.07,Z 405.252,A -85,B 0,C 180,E1 -21230.229,E2 -21230.229} C_VEL
LIN {X 0,Y 207.024,Z 405.322,A -85,B 0,C 180,E1 -21234.154,E2 -21234.154} C_VEL
LIN {X 0,Y 207.313,Z 405.265,A -85,B 0,C 180,E1 -21238.057,E2 -21238.057} C_VEL
LIN {X 0,Y 207.471,Z 405.261,A -85,B 0,C 180,E1 -21240,E2 -21240} C_VEL
LIN {X 0,Y 207.339,Z 405.277,A -85,B 0,C 180,E1 -21241.942,E2 -21241.942} C_VEL
LIN {X 0,Y 207.116,Z 405.302,A -85,B 0,C 180,E1 -21247.8,E2 -21247.8} C_VEL
LIN {X 0,Y 206.898,Z 405.339,A -85,B 0,C 180,E1 -21251.759,E2 -21251.759} C_VEL
LIN {X 0,Y 206.795,Z 405.345,A -85,B 0,C 180,E1 -21255.776,E2 -21255.776} C_VEL
LIN {X 0,Y 206.706,Z 405.355,A -85,B 0,C 180,E1 -21259.876,E2 -21259.876} C_VEL
LIN {X 0,Y 206.694,Z 405.359,A -85,B 0,C 180,E1 -21264.08,E2 -21264.08} C_VEL
LIN {X 0,Y 206.744,Z 405.471,A -85,B 0,C 180,E1 -21267.475,E2 -21267.475} C_VEL
LIN {X 0,Y 210.226,Z 414.875,A -85,B 0,C 180,E1 -21272.336,E2 -21272.336} C_VEL
LIN {X 0,Y 211.822,Z 419.244,A -85,B 0,C 180,E1 -21274.293,E2 -21274.293} C_VEL
LIN {X 0,Y 216.525,Z 427.351,A -85,B 0,C 180,E1 -21276.186,E2 -21276.186} C_VEL
LIN {X 0,Y 220.275,Z 433.996,A -85,B 0,C 180,E1 -21277.603,E2 -21277.603} C_VEL
LIN {X 0,Y 225.182,Z 443.171,A -85,B 0,C 180,E1 -21279.356,E2 -21279.356} C_VEL
LIN {X 0,Y 227.074,Z 448.014,A -85,B 0,C 180,E1 -21280.055,E2 -21280.055} C_VEL
LIN {X 0,Y 228.198,Z 453.478,A -85,B 0,C 180,E1 -21280.573,E2 -21280.573} C_VEL
LIN {X 0,Y 230.107,Z 466.762,A -85,B 0,C 180,E1 -21281.603,E2 -21281.603} C_VEL
LIN {X 0,Y 231.684,Z 472.029,A -85,B 0,C 180,E1 -21282.19,E2 -21282.19} C_VEL
LIN {X 0,Y 233.501,Z 477.076,A -85,B 0,C 180,E1 -21282.809,E2 -21282.809} C_VEL
LIN {X 0,Y 236.982,Z 523.141,A -85,B 0,C 180,E1 -21285.377,E2 -21285.377} C_VEL
LIN {X 0,Y 233.158,Z 592.94,A -85,B 0,C 180,E1 -21287.37,E2 -21287.37} C_VEL
LIN {X 0,Y 231.43,Z 608.496,A -85,B 0,C 180,E1 -21288.081,E2 -21288.081} C_VEL
LIN {X 0,Y 228.856,Z 624.156,A -85,B 0,C 180,E1 -21289.119,E2 -21289.119} C_VEL
LIN {X 0,Y 225.891,Z 638.15,A -85,B 0,C 180,E1 -21290.372,E2 -21290.372} C_VEL
LIN {X 0,Y 222.239,Z 651.819,A -85,B 0,C 180,E1 -21291.928,E2 -21291.928} C_VEL
LIN {X 0,Y 218.184,Z 665.111,A -85,B 0,C 180,E1 -21293.855,E2 -21293.855} C_VEL
LIN {X 0,Y 214.45,Z 677.399,A -85,B 0,C 180,E1 -21296.143,E2 -21296.143} C_VEL
LIN {X 0,Y 210.441,Z 689.15,A -85,B 0,C 180,E1 -21298.825,E2 -21298.825} C_VEL
LIN {X 0,Y 207.042,Z 699.078,A -85,B 0,C 180,E1 -21301.626,E2 -21301.626} C_VEL
LIN {X 0,Y 203.82,Z 708.875,A -85,B 0,C 180,E1 -21305.014,E2 -21305.014} C_VEL
LIN {X 0,Y 201.403,Z 717.068,A -85,B 0,C 180,E1 -21308.506,E2 -21308.506} C_VEL
LIN {X 0,Y 199.536,Z 724.868,A -85,B 0,C 180,E1 -21312.651,E2 -21312.651} C_VEL
LIN {X 0,Y 198.691,Z 730.868,A -85,B 0,C 180,E1 -21316.707,E2 -21316.707} C_VEL
LIN {X 0,Y 198.625,Z 734.544,A -85,B 0,C 180,E1 -21319.809,E2 -21319.809} C_VEL
LIN {X 0,Y 199.117,Z 738.206,A -85,B 0,C 180,E1 -21323.921,E2 -21323.921} C_VEL
LIN {X 0,Y 199.766,Z 740.512,A -85,B 0,C 180,E1 -21327.983,E2 -21327.983} C_VEL
LIN {X 0,Y 200.256,Z 741.196,A -85,B 0,C 180,E1 -21329.999,E2 -21329.999} C_VEL
LIN {X 0,Y 199.243,Z 741.318,A -85,B 0,C 180,E1 -21334.045,E2 -21334.045} C_VEL
LIN {X 0,Y 198.627,Z 740.347,A -85,B 0,C 180,E1 -21337.815,E2 -21337.815} C_VEL
LIN {X 0,Y 198.343,Z 737.895,A -85,B 0,C 180,E1 -21342.274,E2 -21342.274} C_VEL
LIN {X 0,Y 199.097,Z 734.417,A -85,B 0,C 180,E1 -21346.402,E2 -21346.402} C_VEL
LIN {X 0,Y 200.857,Z 729.734,A -85,B 0,C 180,E1 -21350.48,E2 -21350.48} C_VEL
LIN {X 0,Y 203.673,Z 723.748,A -85,B 0,C 180,E1 -21354.46,E2 -21354.46} C_VEL
LIN {X 0,Y 207.464,Z 716.309,A -85,B 0,C 180,E1 -21358.31,E2 -21358.31} C_VEL
LIN {X 0,Y 211.646,Z 708.494,A -85,B 0,C 180,E1 -21361.532,E2 -21361.532} C_VEL
LIN {X 0,Y 216.645,Z 699.19,A -85,B 0,C 180,E1 -21364.588,E2 -21364.588} C_VEL
LIN {X 0,Y 222.362,Z 688.249,A -85,B 0,C 180,E1 -21367.429,E2 -21367.429} C_VEL
LIN {X 0,Y 227.783,Z 676.793,A -85,B 0,C 180,E1 -21369.806,E2 -21369.806} C_VEL
LIN {X 0,Y 233.201,Z 664.48,A -85,B 0,C 180,E1 -21371.817,E2 -21371.817} C_VEL
LIN {X 0,Y 238.583,Z 651.03,A -85,B 0,C 180,E1 -21373.514,E2 -21373.514} C_VEL
LIN {X 0,Y 243.051,Z 637.902,A -85,B 0,C 180,E1 -21374.813,E2 -21374.813} C_VEL
LIN {X 0,Y 246.462,Z 625.909,A -85,B 0,C 180,E1 -21375.76,E2 -21375.76} C_VEL
LIN {X 0,Y 249.886,Z 610.634,A -85,B 0,C 180,E1 -21376.694,E2 -21376.694} C_VEL
LIN {X 0,Y 252.421,Z 594.936,A -85,B 0,C 180,E1 -21377.365,E2 -21377.365} C_VEL
LIN {X 0,Y 254.01,Z 576.783,A -85,B 0,C 180,E1 -21377.9,E2 -21377.9} C_VEL
LIN {X 0,Y 257.325,Z 526.49,A -85,B 0,C 180,E1 -21379.199,E2 -21379.199} C_VEL
LIN {X 0,Y 255.489,Z 498.163,A -85,B 0,C 180,E1 -21381.044,E2 -21381.044} C_VEL
LIN {X 0,Y 252.624,Z 490.759,A -85,B 0,C 180,E1 -21382.311,E2 -21382.311} C_VEL
LIN {X 0,Y 248.014,Z 480.303,A -85,B 0,C 180,E1 -21384.431,E2 -21384.431} C_VEL
LIN {X 0,Y 243.548,Z 470.993,A -85,B 0,C 180,E1 -21386.651,E2 -21386.651} C_VEL
LIN {X 0,Y 240.175,Z 464.412,A -85,B 0,C 180,E1 -21388.463,E2 -21388.463} C_VEL
LIN {X 0,Y 237.178,Z 458.796,A -85,B 0,C 180,E1 -21390.198,E2 -21390.198} C_VEL
LIN {X 0,Y 233.88,Z 452.755,A -85,B 0,C 180,E1 -21392.293,E2 -21392.293} C_VEL
LIN {X 0,Y 229.449,Z 445.119,A -85,B 0,C 180,E1 -21395.485,E2 -21395.485} C_VEL
LIN {X 0,Y 224.356,Z 436.531,A -85,B 0,C 180,E1 -21400.038,E2 -21400.038} C_VEL
LIN {X 0,Y 219.645,Z 428.427,A -85,B 0,C 180,E1 -21406.174,E2 -21406.174} C_VEL
LIN {X 0,Y 218.165,Z 425.773,A -85,B 0,C 180,E1 -21409.179,E2 -21409.179} C_VEL
LIN {X 0,Y 217.76,Z 424.567,A -85,B 0,C 180,E1 -21410.406,E2 -21410.406} C_VEL
LIN {X 0,Y 217.01,Z 424.127,A -85,B 0,C 180,E1 -21420,E2 -21420} C_VEL
LIN {X 0,Y 217.993,Z 424.721,A -85,B 0,C 180,E1 -21423.119,E2 -21423.119} C_VEL
LIN {X 0,Y 219.086,Z 427.252,A -85,B 0,C 180,E1 -21425.754,E2 -21425.754} C_VEL
LIN {X 0,Y 221.844,Z 429.959,A -85,B 0,C 180,E1 -21429.765,E2 -21429.765} C_VEL
LIN {X 0,Y 222.514,Z 430.631,A -85,B 0,C 180,E1 -21430.552,E2 -21430.552} C_VEL
LIN {X 0,Y 224.597,Z 433.984,A -85,B 0,C 180,E1 -21432.883,E2 -21432.883} C_VEL
LIN {X 0,Y 226.69,Z 435.91,A -85,B 0,C 180,E1 -21434.762,E2 -21434.762} C_VEL
LIN {X 0,Y 229.266,Z 439.591,A -85,B 0,C 180,E1 -21436.919,E2 -21436.919} C_VEL
LIN {X 0,Y 230.762,Z 441.244,A -85,B 0,C 180,E1 -21438.018,E2 -21438.018} C_VEL
LIN {X 0,Y 233.706,Z 445.123,A -85,B 0,C 180,E1 -21440.046,E2 -21440.046} C_VEL
LIN {X 0,Y 238.452,Z 451.583,A -85,B 0,C 180,E1 -21442.93,E2 -21442.93} C_VEL
LIN {X 0,Y 241.909,Z 456.502,A -85,B 0,C 180,E1 -21444.807,E2 -21444.807} C_VEL
LIN {X 0,Y 246.708,Z 463.574,A -85,B 0,C 180,E1 -21447.174,E2 -21447.174} C_VEL
LIN {X 0,Y 252.502,Z 472.762,A -85,B 0,C 180,E1 -21449.751,E2 -21449.751} C_VEL
LIN {X 0,Y 259.115,Z 484.48,A -85,B 0,C 180,E1 -21452.419,E2 -21452.419} C_VEL
LIN {X 0,Y 259.858,Z 485.866,A -85,B 0,C 180,E1 -21452.703,E2 -21452.703} C_VEL
LIN {X 0,Y 256.883,Z 535.4,A -85,B 0,C 180,E1 -21454.067,E2 -21454.067} C_VEL
LIN {X 0,Y 255.691,Z 551.1,A -85,B 0,C 180,E1 -21454.686,E2 -21454.686} C_VEL
LIN {X 0,Y 253.948,Z 565.234,A -85,B 0,C 180,E1 -21455.534,E2 -21455.534} C_VEL
LIN {X 0,Y 251.598,Z 577.341,A -85,B 0,C 180,E1 -21456.409,E2 -21456.409} C_VEL
LIN {X 0,Y 248.596,Z 590.514,A -85,B 0,C 180,E1 -21457.669,E2 -21457.669} C_VEL
LIN {X 0,Y 244.849,Z 603.513,A -85,B 0,C 180,E1 -21459.199,E2 -21459.199} C_VEL
LIN {X 0,Y 240.691,Z 615.517,A -85,B 0,C 180,E1 -21460.931,E2 -21460.931} C_VEL
LIN {X 0,Y 236.055,Z 627.217,A -85,B 0,C 180,E1 -21463.035,E2 -21463.035} C_VEL
LIN {X 0,Y 230.881,Z 638.566,A -85,B 0,C 180,E1 -21465.566,E2 -21465.566} C_VEL
LIN {X 0,Y 225.761,Z 648.549,A -85,B 0,C 180,E1 -21468.343,E2 -21468.343} C_VEL
LIN {X 0,Y 220.513,Z 657.754,A -85,B 0,C 180,E1 -21471.577,E2 -21471.577} C_VEL
LIN {X 0,Y 216.657,Z 663.956,A -85,B 0,C 180,E1 -21474.277,E2 -21474.277} C_VEL
LIN {X 0,Y 212.181,Z 670.695,A -85,B 0,C 180,E1 -21477.999,E2 -21477.999} C_VEL
LIN {X 0,Y 208.425,Z 675.896,A -85,B 0,C 180,E1 -21481.833,E2 -21481.833} C_VEL
LIN {X 0,Y 205.422,Z 679.722,A -85,B 0,C 180,E1 -21485.762,E2 -21485.762} C_VEL
LIN {X 0,Y 203.161,Z 682.297,A -85,B 0,C 180,E1 -21489.763,E2 -21489.763} C_VEL
LIN {X 0,Y 201.578,Z 683.709,A -85,B 0,C 180,E1 -21493.806,E2 -21493.806} C_VEL
LIN {X 0,Y 200.732,Z 683.991,A -85,B 0,C 180,E1 -21497.875,E2 -21497.875} C_VEL
LIN {X 0,Y 200.439,Z 683.182,A -85,B 0,C 180,E1 -21501.939,E2 -21501.939} C_VEL
LIN {X 0,Y 200.598,Z 681.246,A -85,B 0,C 180,E1 -21505.983,E2 -21505.983} C_VEL
LIN {X 0,Y 201.462,Z 678.15,A -85,B 0,C 180,E1 -21510.001,E2 -21510.001} C_VEL
LIN {X 0,Y 202.843,Z 673.875,A -85,B 0,C 180,E1 -21513.974,E2 -21513.974} C_VEL
LIN {X 0,Y 204.876,Z 668.299,A -85,B 0,C 180,E1 -21517.887,E2 -21517.887} C_VEL
LIN {X 0,Y 207.519,Z 661.274,A -85,B 0,C 180,E1 -21521.725,E2 -21521.725} C_VEL
LIN {X 0,Y 210.779,Z 652.571,A -85,B 0,C 180,E1 -21525.471,E2 -21525.471} C_VEL
LIN {X 0,Y 214.188,Z 643.303,A -85,B 0,C 180,E1 -21528.658,E2 -21528.658} C_VEL
LIN {X 0,Y 217.416,Z 633.882,A -85,B 0,C 180,E1 -21531.325,E2 -21531.325} C_VEL
LIN {X 0,Y 220.943,Z 622.704,A -85,B 0,C 180,E1 -21533.927,E2 -21533.927} C_VEL
LIN {X 0,Y 223.958,Z 611.709,A -85,B 0,C 180,E1 -21536.061,E2 -21536.061} C_VEL
LIN {X 0,Y 227.393,Z 598.355,A -85,B 0,C 180,E1 -21538.121,E2 -21538.121} C_VEL
LIN {X 0,Y 230.163,Z 585.299,A -85,B 0,C 180,E1 -21539.748,E2 -21539.748} C_VEL
LIN {X 0,Y 232.662,Z 570.858,A -85,B 0,C 180,E1 -21541.151,E2 -21541.151} C_VEL
LIN {X 0,Y 234.57,Z 555.808,A -85,B 0,C 180,E1 -21542.255,E2 -21542.255} C_VEL
LIN {X 0,Y 235.835,Z 540.359,A -85,B 0,C 180,E1 -21543.047,E2 -21543.047} C_VEL
LIN {X 0,Y 237.361,Z 504.663,A -85,B 0,C 180,E1 -21544.179,E2 -21544.179} C_VEL
LIN {X 0,Y 239.2,Z 469.252,A -85,B 0,C 180,E1 -21545.185,E2 -21545.185} C_VEL
LIN {X 0,Y 231.89,Z 454.868,A -85,B 0,C 180,E1 -21547.396,E2 -21547.396} C_VEL
LIN {X 0,Y 224.351,Z 441.784,A -85,B 0,C 180,E1 -21549.841,E2 -21549.841} C_VEL
LIN {X 0,Y 216.593,Z 429.843,A -85,B 0,C 180,E1 -21552.587,E2 -21552.587} C_VEL
LIN {X 0,Y 209.858,Z 420.628,A -85,B 0,C 180,E1 -21555.211,E2 -21555.211} C_VEL
LIN {X 0,Y 207.235,Z 416.876,A -85,B 0,C 180,E1 -21556.33,E2 -21556.33} C_VEL
LIN {X 0,Y 204.401,Z 413.674,A -85,B 0,C 180,E1 -21557.555,E2 -21557.555} C_VEL
LIN {X 0,Y 203.282,Z 411.634,A -85,B 0,C 180,E1 -21558.104,E2 -21558.104} C_VEL
LIN {X 0,Y 200.907,Z 409.552,A -85,B 0,C 180,E1 -21559.177,E2 -21559.177} C_VEL
LIN {X 0,Y 199.758,Z 407.113,A -85,B 0,C 180,E1 -21559.805,E2 -21559.805} C_VEL
LIN {X 0,Y 199.598,Z 406.249,A -85,B 0,C 180,E1 -21559.972,E2 -21559.972} C_VEL
LIN {X 0,Y 199.611,Z 406.249,A -85,B 0,C 180,E1 -21564.075,E2 -21564.075} C_VEL
LIN {X 0,Y 199.684,Z 406.238,A -85,B 0,C 180,E1 -21568.133,E2 -21568.133} C_VEL
LIN {X 0,Y 199.64,Z 406.242,A -85,B 0,C 180,E1 -21572.764,E2 -21572.764} C_VEL
LIN {X 0,Y 199.676,Z 406.229,A -85,B 0,C 180,E1 -21577.221,E2 -21577.221} C_VEL
LIN {X 0,Y 199.744,Z 406.215,A -85,B 0,C 180,E1 -21581.802,E2 -21581.802} C_VEL
LIN {X 0,Y 199.807,Z 406.197,A -85,B 0,C 180,E1 -21585.746,E2 -21585.746} C_VEL
LIN {X 0,Y 200.021,Z 406.127,A -85,B 0,C 180,E1 -21589.881,E2 -21589.881} C_VEL
LIN {X 0,Y 199.989,Z 406.195,A -85,B 0,C 180,E1 -21593.948,E2 -21593.948} C_VEL
LIN {X 0,Y 200.258,Z 406.143,A -85,B 0,C 180,E1 -21597.988,E2 -21597.988} C_VEL
LIN {X 0,Y 200.438,Z 406.137,A -85,B 0,C 180,E1 -21599.999,E2 -21599.999} C_VEL
LIN {X 0,Y 199.982,Z 406.179,A -85,B 0,C 180,E1 -21604.03,E2 -21604.03} C_VEL
LIN {X 0,Y 200.065,Z 406.177,A -85,B 0,C 180,E1 -21608.077,E2 -21608.077} C_VEL
LIN {X 0,Y 199.848,Z 406.216,A -85,B 0,C 180,E1 -21612.18,E2 -21612.18} C_VEL
LIN {X 0,Y 199.736,Z 406.231,A -85,B 0,C 180,E1 -21616.349,E2 -21616.349} C_VEL
LIN {X 0,Y 199.64,Z 406.242,A -85,B 0,C 180,E1 -21620.611,E2 -21620.611} C_VEL
LIN {X 0,Y 199.625,Z 406.242,A -85,B 0,C 180,E1 -21625.199,E2 -21625.199} C_VEL
LIN {X 0,Y 202.156,Z 412.909,A -85,B 0,C 180,E1 -21629.124,E2 -21629.124} C_VEL
LIN {X 0,Y 203.821,Z 417.407,A -85,B 0,C 180,E1 -21631.362,E2 -21631.362} C_VEL
LIN {X 0,Y 208.753,Z 425.344,A -85,B 0,C 180,E1 -21633.587,E2 -21633.587} C_VEL
LIN {X 0,Y 213.195,Z 433.063,A -85,B 0,C 180,E1 -21635.449,E2 -21635.449} C_VEL
LIN {X 0,Y 217.149,Z 440.379,A -85,B 0,C 180,E1 -21637.01,E2 -21637.01} C_VEL
LIN {X 0,Y 221.884,Z 449.663,A -85,B 0,C 180,E1 -21638.778,E2 -21638.778} C_VEL
LIN {X 0,Y 227.844,Z 462.609,A -85,B 0,C 180,E1 -21640.882,E2 -21640.882} C_VEL
LIN {X 0,Y 231.684,Z 472.029,A -85,B 0,C 180,E1 -21642.19,E2 -21642.19} C_VEL
LIN {X 0,Y 232.261,Z 475.004,A -85,B 0,C 180,E1 -21642.445,E2 -21642.445} C_VEL
LIN {X 0,Y 231.809,Z 479.588,A -85,B 0,C 180,E1 -21642.532,E2 -21642.532} C_VEL
LIN {X 0,Y 229.537,Z 489.046,A -85,B 0,C 180,E1 -21642.406,E2 -21642.406} C_VEL
LIN {X 0,Y 229.336,Z 493.154,A -85,B 0,C 180,E1 -21642.532,E2 -21642.532} C_VEL
LIN {X 0,Y 231.518,Z 524.045,A -85,B 0,C 180,E1 -21644.282,E2 -21644.282} C_VEL
LIN {X 0,Y 227.659,Z 591.601,A -85,B 0,C 180,E1 -21646.236,E2 -21646.236} C_VEL
LIN {X 0,Y 225.896,Z 607.295,A -85,B 0,C 180,E1 -21646.96,E2 -21646.96} C_VEL
LIN {X 0,Y 223.267,Z 623.029,A -85,B 0,C 180,E1 -21648.018,E2 -21648.018} C_VEL
LIN {X 0,Y 219.951,Z 637.994,A -85,B 0,C 180,E1 -21649.381,E2 -21649.381} C_VEL
LIN {X 0,Y 216.195,Z 651.525,A -85,B 0,C 180,E1 -21650.962,E2 -21650.962} C_VEL
LIN {X 0,Y 211.968,Z 664.81,A -85,B 0,C 180,E1 -21652.944,E2 -21652.944} C_VEL
LIN {X 0,Y 207.793,Z 677.959,A -85,B 0,C 180,E1 -21655.492,E2 -21655.492} C_VEL
LIN {X 0,Y 203.662,Z 689.459,A -85,B 0,C 180,E1 -21658.248,E2 -21658.248} C_VEL
LIN {X 0,Y 199.603,Z 700.804,A -85,B 0,C 180,E1 -21661.672,E2 -21661.672} C_VEL
LIN {X 0,Y 196.453,Z 710.05,A -85,B 0,C 180,E1 -21665.143,E2 -21665.143} C_VEL
LIN {X 0,Y 194.095,Z 717.881,A -85,B 0,C 180,E1 -21668.771,E2 -21668.771} C_VEL
LIN {X 0,Y 192.31,Z 725.204,A -85,B 0,C 180,E1 -21673,E2 -21673} C_VEL
LIN {X 0,Y 191.575,Z 730.998,A -85,B 0,C 180,E1 -21677.284,E2 -21677.284} C_VEL
LIN {X 0,Y 191.74,Z 735.554,A -85,B 0,C 180,E1 -21681.747,E2 -21681.747} C_VEL
LIN {X 0,Y 192.306,Z 738.419,A -85,B 0,C 180,E1 -21685.808,E2 -21685.808} C_VEL
LIN {X 0,Y 193.216,Z 740.148,A -85,B 0,C 180,E1 -21689.999,E2 -21689.999} C_VEL
LIN {X 0,Y 192.173,Z 740.304,A -85,B 0,C 180,E1 -21694.194,E2 -21694.194} C_VEL
LIN {X 0,Y 191.567,Z 739.416,A -85,B 0,C 180,E1 -21697.887,E2 -21697.887} C_VEL
LIN {X 0,Y 191.318,Z 736.928,A -85,B 0,C 180,E1 -21702.732,E2 -21702.732} C_VEL
LIN {X 0,Y 192.189,Z 733.491,A -85,B 0,C 180,E1 -21707.009,E2 -21707.009} C_VEL
LIN {X 0,Y 194.106,Z 728.854,A -85,B 0,C 180,E1 -21711.226,E2 -21711.226} C_VEL
LIN {X 0,Y 197.118,Z 722.921,A -85,B 0,C 180,E1 -21715.329,E2 -21715.329} C_VEL
LIN {X 0,Y 201.157,Z 715.541,A -85,B 0,C 180,E1 -21719.282,E2 -21719.282} C_VEL
LIN {X 0,Y 206.244,Z 706.518,A -85,B 0,C 180,E1 -21723.038,E2 -21723.038} C_VEL
LIN {X 0,Y 210.794,Z 698.52,A -85,B 0,C 180,E1 -21725.692,E2 -21725.692} C_VEL
LIN {X 0,Y 215.898,Z 689.187,A -85,B 0,C 180,E1 -21728.204,E2 -21728.204} C_VEL
LIN {X 0,Y 221.385,Z 678.266,A -85,B 0,C 180,E1 -21730.599,E2 -21730.599} C_VEL
LIN {X 0,Y 226.898,Z 666.452,A -85,B 0,C 180,E1 -21732.651,E2 -21732.651} C_VEL
LIN {X 0,Y 232.343,Z 653.643,A -85,B 0,C 180,E1 -21734.384,E2 -21734.384} C_VEL
LIN {X 0,Y 237.499,Z 639.61,A -85,B 0,C 180,E1 -21735.854,E2 -21735.854} C_VEL
LIN {X 0,Y 241.576,Z 626.122,A -85,B 0,C 180,E1 -21736.963,E2 -21736.963} C_VEL
LIN {X 0,Y 245.087,Z 611.294,A -85,B 0,C 180,E1 -21737.898,E2 -21737.898} C_VEL
LIN {X 0,Y 247.756,Z 595.979,A -85,B 0,C 180,E1 -21738.582,E2 -21738.582} C_VEL
LIN {X 0,Y 249.384,Z 580.057,A -85,B 0,C 180,E1 -21739.074,E2 -21739.074} C_VEL
LIN {X 0,Y 252.976,Z 527.767,A -85,B 0,C 180,E1 -21740.426,E2 -21740.426} C_VEL
LIN {X 0,Y 251.41,Z 501.265,A -85,B 0,C 180,E1 -21742.192,E2 -21742.192} C_VEL
LIN {X 0,Y 247.266,Z 490.826,A -85,B 0,C 180,E1 -21744.145,E2 -21744.145} C_VEL
LIN {X 0,Y 242.258,Z 479.648,A -85,B 0,C 180,E1 -21746.673,E2 -21746.673} C_VEL
LIN {X 0,Y 237.726,Z 470.34,A -85,B 0,C 180,E1 -21749.19,E2 -21749.19} C_VEL
LIN {X 0,Y 234.68,Z 464.467,A -85,B 0,C 180,E1 -21751.045,E2 -21751.045} C_VEL
LIN {X 0,Y 231.573,Z 458.592,A -85,B 0,C 180,E1 -21753.129,E2 -21753.129} C_VEL
LIN {X 0,Y 227.482,Z 451.238,A -85,B 0,C 180,E1 -21756.245,E2 -21756.245} C_VEL
LIN {X 0,Y 222.788,Z 442.988,A -85,B 0,C 180,E1 -21760.682,E2 -21760.682} C_VEL
LIN {X 0,Y 218.281,Z 434.977,A -85,B 0,C 180,E1 -21766.975,E2 -21766.975} C_VEL
LIN {X 0,Y 217.065,Z 432.433,A -85,B 0,C 180,E1 -21769.757,E2 -21769.757} C_VEL
LIN {X 0,Y 216.786,Z 431.575,A -85,B 0,C 180,E1 -21770.672,E2 -21770.672} C_VEL
LIN {X 0,Y 216.14,Z 431.158,A -85,B 0,C 180,E1 -21780,E2 -21780} C_VEL
LIN {X 0,Y 216.982,Z 431.696,A -85,B 0,C 180,E1 -21782.785,E2 -21782.785} C_VEL
LIN {X 0,Y 218.203,Z 434.423,A -85,B 0,C 180,E1 -21785.777,E2 -21785.777} C_VEL
LIN {X 0,Y 221.201,Z 437.455,A -85,B 0,C 180,E1 -21790.092,E2 -21790.092} C_VEL
LIN {X 0,Y 223.498,Z 441.03,A -85,B 0,C 180,E1 -21792.717,E2 -21792.717} C_VEL
LIN {X 0,Y 225.205,Z 442.703,A -85,B 0,C 180,E1 -21794.299,E2 -21794.299} C_VEL
LIN {X 0,Y 227.902,Z 446.473,A -85,B 0,C 180,E1 -21796.612,E2 -21796.612} C_VEL
LIN {X 0,Y 229.128,Z 447.986,A -85,B 0,C 180,E1 -21797.551,E2 -21797.551} C_VEL
LIN {X 0,Y 232.796,Z 452.973,A -85,B 0,C 180,E1 -21800.128,E2 -21800.128} C_VEL
LIN {X 0,Y 236.699,Z 458.419,A -85,B 0,C 180,E1 -21802.54,E2 -21802.54} C_VEL
LIN {X 0,Y 241.707,Z 465.739,A -85,B 0,C 180,E1 -21805.278,E2 -21805.278} C_VEL
LIN {X 0,Y 247.761,Z 475.317,A -85,B 0,C 180,E1 -21808.208,E2 -21808.208} C_VEL
LIN {X 0,Y 254.042,Z 486.387,A -85,B 0,C 180,E1 -21810.934,E2 -21810.934} C_VEL
LIN {X 0,Y 255.465,Z 489.041,A -85,B 0,C 180,E1 -21811.514,E2 -21811.514} C_VEL
LIN {X 0,Y 252.558,Z 535.348,A -85,B 0,C 180,E1 -21812.797,E2 -21812.797} C_VEL
LIN {X 0,Y 251.45,Z 550.221,A -85,B 0,C 180,E1 -21813.372,E2 -21813.372} C_VEL
LIN {X 0,Y 249.644,Z 564.65,A -85,B 0,C 180,E1 -21814.197,E2 -21814.197} C_VEL
LIN {X 0,Y 247.107,Z 577.893,A -85,B 0,C 180,E1 -21815.15,E2 -21815.15} C_VEL
LIN {X 0,Y 244.242,Z 590.28,A -85,B 0,C 180,E1 -21816.326,E2 -21816.326} C_VEL
LIN {X 0,Y 240.267,Z 603.781,A -85,B 0,C 180,E1 -21817.899,E2 -21817.899} C_VEL
LIN {X 0,Y 236.046,Z 615.711,A -85,B 0,C 180,E1 -21819.613,E2 -21819.613} C_VEL
LIN {X 0,Y 231.04,Z 627.872,A -85,B 0,C 180,E1 -21821.792,E2 -21821.792} C_VEL
LIN {X 0,Y 225.796,Z 639.018,A -85,B 0,C 180,E1 -21824.287,E2 -21824.287} C_VEL
LIN {X 0,Y 220.983,Z 648.096,A -85,B 0,C 180,E1 -21826.793,E2 -21826.793} C_VEL
LIN {X 0,Y 215.619,Z 657.247,A -85,B 0,C 180,E1 -21829.931,E2 -21829.931} C_VEL
LIN {X 0,Y 210.87,Z 664.627,A -85,B 0,C 180,E1 -21833.138,E2 -21833.138} C_VEL
LIN {X 0,Y 206.111,Z 671.44,A -85,B 0,C 180,E1 -21836.938,E2 -21836.938} C_VEL
LIN {X 0,Y 202.109,Z 676.709,A -85,B 0,C 180,E1 -21840.87,E2 -21840.87} C_VEL
LIN {X 0,Y 198.9,Z 680.595,A -85,B 0,C 180,E1 -21844.913,E2 -21844.913} C_VEL
LIN {X 0,Y 196.446,Z 683.23,A -85,B 0,C 180,E1 -21849.039,E2 -21849.039} C_VEL
LIN {X 0,Y 194.717,Z 684.697,A -85,B 0,C 180,E1 -21853.218,E2 -21853.218} C_VEL
LIN {X 0,Y 193.777,Z 685.031,A -85,B 0,C 180,E1 -21857.432,E2 -21857.432} C_VEL
LIN {X 0,Y 193.434,Z 684.254,A -85,B 0,C 180,E1 -21861.645,E2 -21861.645} C_VEL
LIN {X 0,Y 193.542,Z 682.364,A -85,B 0,C 180,E1 -21865.836,E2 -21865.836} C_VEL
LIN {X 0,Y 194.405,Z 679.325,A -85,B 0,C 180,E1 -21870.001,E2 -21870.001} C_VEL
LIN {X 0,Y 195.482,Z 676.305,A -85,B 0,C 180,E1 -21873.092,E2 -21873.092} C_VEL
LIN {X 0,Y 197.357,Z 671.124,A -85,B 0,C 180,E1 -21877.16,E2 -21877.16} C_VEL
LIN {X 0,Y 199.949,Z 664.54,A -85,B 0,C 180,E1 -21881.147,E2 -21881.147} C_VEL
LIN {X 0,Y 203.152,Z 656.375,A -85,B 0,C 180,E1 -21885.038,E2 -21885.038} C_VEL
LIN {X 0,Y 206.529,Z 647.652,A -85,B 0,C 180,E1 -21888.347,E2 -21888.347} C_VEL
LIN {X 0,Y 210.375,Z 637.193,A -85,B 0,C 180,E1 -21891.56,E2 -21891.56} C_VEL
LIN {X 0,Y 213.991,Z 626.434,A -85,B 0,C 180,E1 -21894.238,E2 -21894.238} C_VEL
LIN {X 0,Y 217.394,Z 614.726,A -85,B 0,C 180,E1 -21896.651,E2 -21896.651} C_VEL
LIN {X 0,Y 220.906,Z 601.837,A -85,B 0,C 180,E1 -21898.763,E2 -21898.763} C_VEL
LIN {X 0,Y 223.754,Z 589.297,A -85,B 0,C 180,E1 -21900.429,E2 -21900.429} C_VEL
LIN {X 0,Y 226.382,Z 575.675,A -85,B 0,C 180,E1 -21901.854,E2 -21901.854} C_VEL
LIN {X 0,Y 228.59,Z 560.469,A -85,B 0,C 180,E1 -21903.074,E2 -21903.074} C_VEL
LIN {X 0,Y 230.056,Z 545.302,A -85,B 0,C 180,E1 -21903.949,E2 -21903.949} C_VEL
LIN {X 0,Y 230.972,Z 525.607,A -85,B 0,C 180,E1 -21904.688,E2 -21904.688} C_VEL
LIN {X 0,Y 233.777,Z 471.7,A -85,B 0,C 180,E1 -21906.266,E2 -21906.266} C_VEL
LIN {X 0,Y 226.335,Z 457.049,A -85,B 0,C 180,E1 -21908.649,E2 -21908.649} C_VEL
LIN {X 0,Y 219.406,Z 445.062,A -85,B 0,C 180,E1 -21911.035,E2 -21911.035} C_VEL
LIN {X 0,Y 212.616,Z 434.684,A -85,B 0,C 180,E1 -21913.569,E2 -21913.569} C_VEL
LIN {X 0,Y 206.678,Z 426.329,A -85,B 0,C 180,E1 -21916.003,E2 -21916.003} C_VEL
LIN {X 0,Y 203.576,Z 422.101,A -85,B 0,C 180,E1 -21917.378,E2 -21917.378} C_VEL
LIN {X 0,Y 200.837,Z 418.456,A -85,B 0,C 180,E1 -21918.661,E2 -21918.661} C_VEL
LIN {X 0,Y 199.688,Z 417.162,A -85,B 0,C 180,E1 -21919.208,E2 -21919.208} C_VEL
